C09108=1072.205,-104.494,443.420,172.641,21.693,153.924
C09109=1072.212,-104.245,443.411,172.643,21.694,153.924
C09110=1072.217,-103.995,443.400,172.644,21.695,153.924
C09111=1072.223,-103.745,443.390,172.646,21.696,153.924
C09112=1072.230,-103.495,443.381,172.648,21.697,153.924
C09113=1072.236,-103.246,443.370,172.649,21.699,153.924
C09114=1072.242,-102.996,443.360,172.651,21.700,153.924
C09115=1072.248,-102.746,443.351,172.652,21.701,153.924
C09116=1072.254,-102.497,443.340,172.654,21.702,153.924
C09117=1072.260,-102.247,443.330,172.656,21.704,153.924
C09118=1072.266,-101.997,443.321,172.657,21.705,153.924
C09119=1072.272,-101.748,443.310,172.659,21.706,153.924
C09120=1072.278,-101.498,443.301,172.660,21.708,153.924
C09121=1072.284,-101.249,443.290,172.662,21.709,153.924
C09122=1072.290,-100.999,443.280,172.663,21.710,153.924
C09123=1072.297,-100.748,443.270,172.664,21.711,153.924
C09124=1072.303,-100.499,443.259,172.666,21.712,153.924
C09125=1072.309,-100.249,443.250,172.668,21.714,153.924
C09126=1072.316,-100.000,443.240,172.669,21.715,153.924
C09127=1072.321,-99.750,443.229,172.671,21.716,153.924
C09128=1072.327,-99.500,443.220,172.672,21.717,153.924
C09129=1072.334,-99.251,443.210,172.674,21.719,153.924
C09130=1072.339,-99.001,443.199,172.676,21.720,153.924
C09131=1072.346,-98.752,443.189,172.677,21.721,153.924
C09132=1072.352,-98.501,443.179,172.679,21.722,153.924
C09133=1072.359,-98.220,443.167,172.681,21.724,153.924
C09134=1072.365,-97.938,443.156,172.683,21.726,153.924
C09135=1072.373,-97.657,443.145,172.685,21.727,153.924
C09136=1072.379,-97.374,443.133,172.686,21.728,153.924
C09137=1072.386,-97.125,443.123,172.688,21.730,153.924
C09138=1072.391,-96.875,443.113,172.689,21.731,153.924
C09139=1072.397,-96.626,443.102,172.691,21.733,153.924
C09140=1072.403,-96.376,443.093,172.692,21.734,153.924
C09141=1072.409,-96.126,443.082,172.694,21.735,153.924
C09142=1072.415,-95.877,443.071,172.696,21.737,153.924
C09143=1072.421,-95.626,443.061,172.697,21.738,153.924
C09144=1072.428,-95.377,443.051,172.699,21.739,153.924
C09145=1072.433,-95.127,443.040,172.700,21.741,153.924
C09146=1072.440,-94.878,443.030,172.702,21.742,153.924
C09147=1072.445,-94.628,443.020,172.703,21.744,153.924
C09148=1072.452,-94.379,443.010,172.705,21.745,153.924
C09149=1072.457,-94.128,443.000,172.707,21.746,153.924
C09150=1072.464,-93.879,442.989,172.708,21.748,153.924
C09151=1072.470,-93.629,442.978,172.710,21.749,153.924
C09152=1072.475,-93.379,442.968,172.711,21.751,153.924
C09153=1072.482,-93.130,442.958,172.713,21.753,153.924
C09154=1072.487,-92.880,442.947,172.714,21.754,153.924
C09155=1072.494,-92.630,442.937,172.716,21.755,153.924
C09156=1072.500,-92.381,442.926,172.717,21.757,153.924
C09157=1072.506,-92.131,442.917,172.719,21.758,153.924
C09158=1072.512,-91.881,442.905,172.721,21.759,153.924
C09159=1072.518,-91.631,442.895,172.722,21.761,153.924
C09160=1072.524,-91.382,442.885,172.724,21.762,153.924
C09161=1072.530,-91.132,442.874,172.725,21.764,153.924
C09162=1072.536,-90.882,442.865,172.727,21.765,153.924
C09163=1072.542,-90.632,442.853,172.728,21.766,153.924
C09164=1072.548,-90.383,442.842,172.730,21.768,153.924
C09165=1072.554,-90.133,442.833,172.731,21.770,153.924
C09166=1072.560,-89.883,442.822,172.733,21.771,153.924
C09167=1072.566,-89.634,442.812,172.735,21.773,153.924
C09168=1072.573,-89.384,442.800,172.736,21.774,153.924
C09169=1072.578,-89.134,442.790,172.738,21.775,153.924
C09170=1072.585,-88.885,442.780,172.739,21.777,153.924
C09171=1072.590,-88.635,442.769,172.741,21.778,153.924
C09172=1072.597,-88.386,442.760,172.742,21.780,153.925
C09173=1072.603,-88.135,442.748,172.744,21.781,153.925
C09174=1072.609,-87.886,442.737,172.745,21.783,153.925
C09175=1072.615,-87.637,442.727,172.747,21.784,153.925
C09176=1072.621,-87.387,442.717,172.748,21.786,153.925
C09177=1072.628,-87.137,442.706,172.750,21.787,153.925
C09178=1072.633,-86.887,442.695,172.751,21.789,153.925
C09179=1072.639,-86.638,442.685,172.753,21.790,153.925
C09180=1072.646,-86.389,442.674,172.755,21.792,153.925
C09181=1072.652,-86.138,442.664,172.756,21.793,153.925
C09182=1072.657,-85.888,442.653,172.758,21.794,153.925
C09183=1072.664,-85.639,442.643,172.759,21.796,153.925
C09184=1072.670,-85.389,442.631,172.761,21.798,153.925
C09185=1072.676,-85.139,442.620,172.762,21.799,153.925
C09186=1072.682,-84.890,442.611,172.764,21.801,153.925
C09187=1072.688,-84.640,442.600,172.765,21.802,153.925
C09188=1072.694,-84.390,442.589,172.767,21.804,153.925
C09189=1072.701,-84.141,442.579,172.768,21.805,153.925
C09190=1072.706,-83.891,442.568,172.770,21.807,153.925
C09191=1072.713,-83.641,442.556,172.772,21.808,153.925
C09192=1072.719,-83.392,442.546,172.773,21.809,153.925
C09193=1072.725,-83.142,442.536,172.774,21.811,153.926
C09194=1072.731,-82.892,442.525,172.776,21.813,153.926
C09195=1072.737,-82.642,442.514,172.778,21.814,153.926
C09196=1072.743,-82.393,442.504,172.779,21.816,153.926
C09197=1072.750,-82.113,442.492,172.781,21.817,153.926
C09198=1072.758,-81.834,442.480,172.783,21.819,153.926
C09199=1072.764,-81.554,442.467,172.784,21.821,153.926
C09200=1072.771,-81.275,442.455,172.786,21.823,153.926
C09201=1072.777,-81.026,442.444,172.788,21.824,153.926
C09202=1072.784,-80.776,442.434,172.789,21.826,153.926
C09203=1072.790,-80.526,442.423,172.791,21.827,153.926
C09204=1072.795,-80.277,442.412,172.792,21.829,153.926
C09205=1072.802,-80.027,442.401,172.793,21.831,153.926
C09206=1072.808,-79.778,442.390,172.795,21.832,153.926
C09207=1072.814,-79.527,442.380,172.797,21.833,153.926
C09208=1072.820,-79.277,442.369,172.798,21.835,153.926
C09209=1072.826,-79.028,442.358,172.800,21.837,153.926
C09210=1072.832,-78.778,442.347,172.801,21.839,153.927
C09211=1072.838,-78.528,442.336,172.803,21.840,153.927
C09212=1072.844,-78.279,442.325,172.804,21.842,153.927
C09213=1072.850,-78.030,442.313,172.805,21.843,153.927
C09214=1072.857,-77.780,442.303,172.807,21.845,153.927
C09215=1072.862,-77.530,442.292,172.809,21.847,153.927
C09216=1072.869,-77.280,442.281,172.811,21.848,153.927
C09217=1072.875,-77.031,442.270,172.812,21.850,153.927
C09218=1072.880,-76.781,442.259,172.814,21.852,153.927
C09219=1072.887,-76.531,442.248,172.815,21.854,153.927
C09220=1072.892,-76.281,442.237,172.817,21.855,153.927
C09221=1072.898,-76.032,442.226,172.818,21.857,153.927
C09222=1072.904,-75.782,442.215,172.820,21.858,153.927
C09223=1072.910,-75.532,442.204,172.821,21.860,153.928
C09224=1072.917,-75.282,442.193,172.823,21.862,153.928
C09225=1072.923,-75.033,442.182,172.824,21.864,153.928
C09226=1072.929,-74.783,442.171,172.826,21.865,153.928
C09227=1072.935,-74.534,442.159,172.827,21.867,153.928
C09228=1072.941,-74.284,442.149,172.829,21.868,153.928
C09229=1072.947,-74.034,442.137,172.830,21.870,153.928
C09230=1072.953,-73.785,442.126,172.832,21.872,153.928
C09231=1072.959,-73.535,442.116,172.833,21.874,153.928
C09232=1072.965,-73.285,442.104,172.835,21.875,153.928
C09233=1072.970,-73.035,442.093,172.836,21.877,153.928
C09234=1072.976,-72.786,442.081,172.837,21.879,153.929
C09235=1072.983,-72.536,442.070,172.839,21.880,153.929
C09236=1072.988,-72.287,442.059,172.840,21.882,153.929
C09237=1072.994,-72.037,442.048,172.842,21.884,153.929
C09238=1073.000,-71.787,442.037,172.843,21.886,153.929
C09239=1073.007,-71.538,442.025,172.845,21.888,153.929
C09240=1073.012,-71.288,442.014,172.847,21.890,153.929
C09241=1073.018,-71.038,442.003,172.848,21.891,153.929
C09242=1073.024,-70.789,441.992,172.850,21.893,153.929
C09243=1073.030,-70.538,441.981,172.851,21.895,153.930
C09244=1073.036,-70.290,441.969,172.853,21.897,153.930
C09245=1073.042,-70.039,441.958,172.854,21.898,153.930
C09246=1073.048,-69.790,441.947,172.856,21.900,153.930
C09247=1073.053,-69.540,441.935,172.857,21.902,153.930
C09248=1073.060,-69.291,441.923,172.859,21.904,153.930
C09249=1073.065,-69.041,441.913,172.860,21.906,153.930
C09250=1073.072,-68.791,441.901,172.861,21.908,153.930
C09251=1073.078,-68.542,441.890,172.863,21.909,153.930
C09252=1073.084,-68.292,441.878,172.864,21.911,153.930
C09253=1073.089,-68.042,441.867,172.866,21.913,153.931
C09254=1073.095,-67.792,441.856,172.867,21.914,153.931
C09255=1073.102,-67.543,441.844,172.869,21.916,153.931
C09256=1073.107,-67.293,441.833,172.870,21.918,153.931
C09257=1073.114,-67.043,441.822,172.871,21.920,153.931
C09258=1073.119,-66.794,441.810,172.873,21.921,153.931
C09259=1073.125,-66.544,441.799,172.875,21.924,153.931
C09260=1073.131,-66.295,441.787,172.877,21.926,153.931
C09261=1073.138,-66.018,441.774,172.878,21.928,153.932
C09262=1073.145,-65.740,441.762,172.879,21.930,153.932
C09263=1073.152,-65.463,441.750,172.881,21.931,153.932
C09264=1073.158,-65.185,441.736,172.883,21.934,153.932
C09265=1073.164,-64.937,441.725,172.885,21.935,153.932
C09266=1073.170,-64.686,441.714,172.886,21.937,153.932
C09267=1073.176,-64.438,441.702,172.887,21.939,153.932
C09268=1073.182,-64.187,441.690,172.889,21.941,153.932
C09269=1073.188,-63.937,441.679,172.890,21.943,153.933
C09270=1073.194,-63.688,441.667,172.892,21.944,153.933
C09271=1073.200,-63.438,441.656,172.893,21.946,153.933
C09272=1073.206,-63.189,441.644,172.895,21.948,153.933
C09273=1073.212,-62.938,441.633,172.896,21.950,153.933
C09274=1073.218,-62.689,441.621,172.897,21.952,153.933
C09275=1073.224,-62.439,441.610,172.899,21.953,153.933
C09276=1073.230,-62.190,441.598,172.900,21.955,153.933
C09277=1073.236,-61.940,441.586,172.903,21.958,153.933
C09278=1073.242,-61.691,441.575,172.904,21.960,153.934
C09279=1073.248,-61.441,441.564,172.905,21.962,153.934
C09280=1073.254,-61.192,441.552,172.907,21.963,153.934
C09281=1073.260,-60.941,441.540,172.908,21.965,153.934
C09282=1073.267,-60.692,441.528,172.910,21.967,153.934
C09283=1073.272,-60.442,441.517,172.911,21.969,153.934
C09284=1073.279,-60.193,441.505,172.912,21.971,153.934
C09285=1073.284,-59.943,441.494,172.914,21.973,153.935
C09286=1073.291,-59.693,441.482,172.915,21.974,153.935
C09287=1073.297,-59.443,441.471,172.917,21.976,153.935
C09288=1073.302,-59.194,441.458,172.918,21.978,153.935
C09289=1073.309,-58.944,441.447,172.920,21.980,153.935
C09290=1073.315,-58.695,441.436,172.921,21.982,153.935
C09291=1073.321,-58.445,441.424,172.923,21.984,153.935
C09292=1073.327,-58.195,441.412,172.925,21.986,153.935
C09293=1073.333,-57.946,441.400,172.926,21.987,153.935
C09294=1073.339,-57.696,441.389,172.928,21.989,153.936
C09295=1073.345,-57.446,441.376,172.929,21.991,153.936
C09296=1073.351,-57.197,441.365,172.930,21.993,153.936
C09297=1073.358,-56.947,441.354,172.932,21.995,153.936
C09298=1073.363,-56.698,441.341,172.933,21.997,153.936
C09299=1073.369,-56.448,441.330,172.935,21.999,153.936
C09300=1073.376,-56.198,441.318,172.936,22.001,153.937
C09301=1073.382,-55.949,441.307,172.937,22.002,153.937
C09302=1073.388,-55.699,441.295,172.939,22.004,153.937
C09303=1073.394,-55.449,441.283,172.940,22.006,153.937
C09304=1073.400,-55.200,441.271,172.942,22.008,153.937
C09305=1073.406,-54.950,441.259,172.944,22.010,153.937
C09306=1073.413,-54.700,441.247,172.945,22.012,153.937
C09307=1073.419,-54.451,441.236,172.947,22.014,153.937
C09308=1073.425,-54.201,441.223,172.948,22.016,153.938
C09309=1073.431,-53.951,441.212,172.949,22.018,153.938
C09310=1073.438,-53.702,441.200,172.951,22.020,153.938
C09311=1073.443,-53.452,441.188,172.952,22.022,153.938
C09312=1073.449,-53.202,441.177,172.954,22.024,153.938
C09313=1073.456,-52.953,441.165,172.955,22.025,153.938
C09314=1073.461,-52.703,441.153,172.957,22.027,153.938
C09315=1073.468,-52.454,441.141,172.958,22.029,153.939
C09316=1073.473,-52.203,441.129,172.959,22.031,153.939
C09317=1073.480,-51.954,441.117,172.962,22.033,153.939
C09318=1073.486,-51.705,441.105,172.963,22.035,153.939
C09319=1073.492,-51.455,441.093,172.964,22.037,153.939
C09320=1073.499,-51.206,441.081,172.966,22.039,153.939
C09321=1073.505,-50.955,441.069,172.967,22.041,153.939
C09322=1073.510,-50.706,441.057,172.969,22.043,153.940
C09323=1073.517,-50.457,441.045,172.970,22.045,153.940
C09324=1073.523,-50.207,441.033,172.971,22.047,153.940
C09325=1073.529,-49.931,441.020,172.973,22.049,153.940
C09326=1073.536,-49.655,441.006,172.975,22.052,153.940
C09327=1073.543,-49.379,440.993,172.976,22.054,153.940
C09328=1073.549,-49.103,440.979,172.978,22.056,153.941
C09329=1073.555,-48.854,440.967,172.979,22.058,153.941
C09330=1073.561,-48.604,440.956,172.981,22.060,153.941
C09331=1073.567,-48.354,440.944,172.983,22.062,153.941
C09332=1073.573,-48.105,440.931,172.984,22.064,153.941
C09333=1073.579,-47.855,440.919,172.985,22.066,153.941
C09334=1073.585,-47.605,440.907,172.987,22.068,153.942
C09335=1073.591,-47.356,440.894,172.988,22.070,153.942
C09336=1073.597,-47.106,440.882,172.989,22.072,153.942
C09337=1073.603,-46.857,440.870,172.991,22.074,153.942
C09338=1073.609,-46.607,440.858,172.992,22.076,153.942
C09339=1073.614,-46.358,440.845,172.993,22.078,153.942
C09340=1073.621,-46.108,440.833,172.995,22.080,153.943
C09341=1073.627,-45.858,440.821,172.997,22.083,153.943
C09342=1073.633,-45.608,440.809,172.998,22.085,153.943
C09343=1073.639,-45.359,440.797,173.000,22.087,153.943
C09344=1073.644,-45.109,440.785,173.001,22.089,153.943
C09345=1073.650,-44.859,440.772,173.003,22.091,153.943
C09346=1073.657,-44.610,440.760,173.004,22.093,153.944
C09347=1073.662,-44.360,440.748,173.005,22.095,153.944
C09348=1073.668,-44.111,440.736,173.007,22.097,153.944
C09349=1073.675,-43.861,440.724,173.008,22.099,153.944
C09350=1073.681,-43.611,440.711,173.009,22.101,153.944
C09351=1073.687,-43.361,440.699,173.012,22.103,153.944
C09352=1073.692,-43.112,440.686,173.013,22.106,153.945
C09353=1073.699,-42.862,440.674,173.014,22.108,153.945
C09354=1073.705,-42.613,440.661,173.016,22.110,153.945
C09355=1073.711,-42.363,440.649,173.017,22.112,153.945
C09356=1073.717,-42.114,440.637,173.018,22.113,153.945
C09357=1073.723,-41.865,440.624,173.020,22.116,153.946
C09358=1073.729,-41.615,440.612,173.021,22.118,153.946
C09359=1073.735,-41.365,440.599,173.022,22.120,153.946
C09360=1073.741,-41.115,440.587,173.024,22.122,153.946
C09361=1073.747,-40.865,440.575,173.026,22.124,153.946
C09362=1073.752,-40.616,440.563,173.027,22.126,153.947
C09363=1073.759,-40.367,440.551,173.029,22.128,153.947
C09364=1073.765,-40.117,440.538,173.030,22.130,153.947
C09365=1073.771,-39.867,440.525,173.031,22.132,153.947
C09366=1073.777,-39.618,440.512,173.033,22.135,153.947
C09367=1073.784,-39.368,440.500,173.034,22.137,153.947
C09368=1073.790,-39.118,440.488,173.035,22.139,153.948
C09369=1073.795,-38.869,440.476,173.037,22.140,153.948
C09370=1073.801,-38.619,440.463,173.038,22.143,153.948
C09371=1073.807,-38.369,440.451,173.040,22.145,153.948
C09372=1073.814,-38.120,440.438,173.042,22.147,153.948
C09373=1073.820,-37.870,440.425,173.043,22.150,153.949
C09374=1073.826,-37.620,440.413,173.044,22.152,153.949
C09375=1073.831,-37.371,440.401,173.046,22.154,153.949
C09376=1073.837,-37.121,440.388,173.047,22.156,153.949
C09377=1073.843,-36.872,440.375,173.048,22.158,153.949
C09378=1073.849,-36.622,440.362,173.050,22.160,153.949
C09379=1073.855,-36.372,440.350,173.051,22.162,153.950
C09380=1073.861,-36.122,440.337,173.053,22.165,153.950
C09381=1073.866,-35.873,440.325,173.054,22.167,153.950
C09382=1073.872,-35.624,440.312,173.056,22.169,153.950
C09383=1073.878,-35.374,440.299,173.057,22.171,153.950
C09384=1073.884,-35.124,440.287,173.058,22.173,153.951
C09385=1073.890,-34.875,440.273,173.060,22.175,153.951
C09386=1073.896,-34.625,440.261,173.061,22.177,153.951
C09387=1073.903,-34.375,440.249,173.062,22.180,153.951
C09388=1073.909,-34.126,440.236,173.064,22.182,153.951
C09389=1073.915,-33.851,440.221,173.066,22.185,153.952
C09390=1073.922,-33.575,440.208,173.067,22.186,153.952
C09391=1073.928,-33.300,440.194,173.068,22.189,153.952
C09392=1073.935,-33.024,440.180,173.071,22.192,153.952
C09393=1073.941,-32.775,440.167,173.072,22.194,153.953
C09394=1073.947,-32.525,440.154,173.073,22.196,153.953
C09395=1073.953,-32.275,440.142,173.075,22.198,153.953
C09396=1073.959,-32.026,440.128,173.076,22.200,153.953
C09397=1073.965,-31.776,440.116,173.077,22.203,153.953
C09398=1073.971,-31.526,440.103,173.079,22.204,153.954
C09399=1073.977,-31.277,440.090,173.081,22.207,153.954
C09400=1073.983,-31.027,440.077,173.082,22.209,153.954
C09401=1073.989,-30.777,440.065,173.083,22.211,153.954
C09402=1073.995,-30.528,440.052,173.085,22.214,153.954
C09403=1074.001,-30.278,440.039,173.086,22.216,153.955
C09404=1074.007,-30.029,440.026,173.087,22.218,153.955
C09405=1074.013,-29.779,440.013,173.089,22.220,153.955
C09406=1074.019,-29.530,440.000,173.090,22.222,153.955
C09407=1074.024,-29.280,439.988,173.091,22.224,153.955
C09408=1074.030,-29.030,439.975,173.094,22.227,153.956
C09409=1074.037,-28.781,439.962,173.095,22.229,153.956
C09410=1074.042,-28.531,439.949,173.096,22.231,153.956
C09411=1074.049,-28.282,439.936,173.097,22.233,153.956
C09412=1074.055,-28.032,439.924,173.099,22.235,153.956
C09413=1074.061,-27.783,439.910,173.100,22.238,153.957
C09414=1074.067,-27.533,439.898,173.101,22.240,153.957
C09415=1074.073,-27.284,439.885,173.103,22.242,153.957
C09416=1074.079,-27.034,439.872,173.104,22.244,153.957
C09417=1074.084,-26.784,439.858,173.106,22.246,153.957
C09418=1074.090,-26.534,439.846,173.108,22.249,153.958
C09419=1074.096,-26.285,439.832,173.109,22.251,153.958
C09420=1074.102,-26.035,439.820,173.110,22.253,153.958
C09421=1074.109,-25.786,439.806,173.111,22.256,153.958
C09422=1074.114,-25.536,439.793,173.113,22.258,153.959
C09423=1074.120,-25.287,439.780,173.114,22.260,153.959
C09424=1074.126,-25.037,439.767,173.115,22.262,153.959
C09425=1074.132,-24.787,439.754,173.117,22.265,153.959
C09426=1074.138,-24.538,439.740,173.119,22.267,153.959
C09427=1074.143,-24.288,439.728,173.120,22.269,153.960
C09428=1074.150,-24.039,439.715,173.121,22.272,153.960
C09429=1074.156,-23.789,439.701,173.123,22.274,153.960
C09430=1074.162,-23.540,439.689,173.124,22.276,153.960
C09431=1074.167,-23.290,439.675,173.125,22.278,153.961
C09432=1074.173,-23.040,439.662,173.127,22.281,153.961
C09433=1074.179,-22.791,439.649,173.129,22.283,153.961
C09434=1074.186,-22.542,439.636,173.130,22.285,153.961
C09435=1074.191,-22.291,439.623,173.131,22.288,153.962
C09436=1074.197,-22.042,439.609,173.133,22.290,153.962
C09437=1074.203,-21.793,439.596,173.134,22.292,153.962
C09438=1074.208,-21.543,439.583,173.135,22.294,153.962
C09439=1074.215,-21.293,439.569,173.137,22.297,153.963
C09440=1074.221,-21.043,439.556,173.138,22.298,153.963
C09441=1074.227,-20.794,439.543,173.140,22.301,153.963
C09442=1074.233,-20.544,439.530,173.141,22.304,153.963
C09443=1074.239,-20.295,439.516,173.143,22.306,153.963
C09444=1074.245,-20.045,439.504,173.144,22.308,153.964
C09445=1074.251,-19.796,439.491,173.145,22.310,153.964
C09446=1074.257,-19.546,439.477,173.146,22.313,153.964
C09447=1074.263,-19.297,439.463,173.148,22.315,153.964
C09448=1074.269,-19.047,439.451,173.149,22.317,153.965
C09449=1074.274,-18.797,439.437,173.151,22.320,153.965
C09450=1074.280,-18.548,439.424,173.153,22.322,153.965
C09451=1074.287,-18.299,439.410,173.154,22.324,153.965
C09452=1074.292,-18.048,439.397,173.155,22.327,153.965
C09453=1074.299,-17.772,439.382,173.156,22.329,153.966
C09454=1074.306,-17.496,439.367,173.159,22.331,153.966
C09455=1074.313,-17.219,439.353,173.160,22.334,153.966
C09456=1074.319,-16.943,439.338,173.161,22.336,153.966
C09457=1074.325,-16.694,439.325,173.162,22.339,153.967
C09458=1074.331,-16.444,439.311,173.165,22.341,153.967
C09459=1074.337,-16.195,439.298,173.166,22.344,153.967
C09460=1074.343,-15.946,439.284,173.167,22.346,153.967
C09461=1074.349,-15.695,439.270,173.168,22.348,153.968
C09462=1074.355,-15.445,439.258,173.170,22.350,153.968
C09463=1074.362,-15.196,439.244,173.171,22.352,153.968
C09464=1074.367,-14.947,439.231,173.172,22.355,153.968
C09465=1074.373,-14.697,439.217,173.174,22.358,153.969
C09466=1074.379,-14.448,439.203,173.176,22.360,153.969
C09467=1074.385,-14.198,439.190,173.177,22.362,153.969
C09468=1074.390,-13.949,439.176,173.178,22.364,153.969
C09469=1074.397,-13.699,439.163,173.179,22.367,153.970
C09470=1074.403,-13.449,439.149,173.181,22.369,153.970
C09471=1074.409,-13.199,439.136,173.182,22.371,153.970
C09472=1074.414,-12.950,439.122,173.183,22.374,153.970
C09473=1074.420,-12.701,439.109,173.185,22.377,153.971
C09474=1074.426,-12.451,439.095,173.187,22.379,153.971
C09475=1074.432,-12.202,439.082,173.188,22.381,153.971
C09476=1074.438,-11.952,439.068,173.189,22.383,153.971
C09477=1074.444,-11.702,439.054,173.191,22.385,153.971
C09478=1074.450,-11.453,439.041,173.192,22.388,153.972
C09479=1074.455,-11.203,439.027,173.193,22.390,153.972
C09480=1074.461,-10.954,439.013,173.195,22.393,153.972
C09481=1074.467,-10.704,439.000,173.197,22.395,153.972
C09482=1074.474,-10.454,438.986,173.198,22.397,153.973
C09483=1074.479,-10.205,438.972,173.199,22.400,153.973
C09484=1074.485,-9.955,438.959,173.200,22.402,153.973
C09485=1074.491,-9.706,438.945,173.202,22.404,153.973
C09486=1074.497,-9.457,438.932,173.203,22.407,153.974
C09487=1074.503,-9.206,438.917,173.204,22.409,153.974
C09488=1074.509,-8.957,438.904,173.206,22.412,153.974
C09489=1074.515,-8.708,438.890,173.208,22.414,153.974
C09490=1074.520,-8.458,438.876,173.209,22.416,153.975
C09491=1074.527,-8.209,438.863,173.210,22.419,153.975
C09492=1074.533,-7.959,438.848,173.211,22.421,153.975
C09493=1074.539,-7.710,438.835,173.213,22.423,153.975
C09494=1074.545,-7.460,438.821,173.214,22.426,153.976
C09495=1074.550,-7.211,438.807,173.216,22.429,153.976
C09496=1074.557,-6.961,438.794,173.217,22.431,153.976
C09497=1074.562,-6.711,438.780,173.219,22.433,153.976
C09498=1074.569,-6.462,438.766,173.220,22.435,153.977
C09499=1074.574,-6.212,438.753,173.221,22.438,153.977
C09500=1074.580,-5.962,438.738,173.223,22.440,153.977
C09501=1074.587,-5.713,438.724,173.224,22.442,153.977
C09502=1074.592,-5.464,438.711,173.226,22.445,153.978
C09503=1074.598,-5.214,438.697,173.227,22.447,153.978
C09504=1074.604,-4.964,438.683,173.228,22.449,153.978
C09505=1074.610,-4.715,438.669,173.230,22.452,153.978
C09506=1074.616,-4.465,438.656,173.231,22.454,153.979
C09507=1074.623,-4.216,438.641,173.232,22.457,153.979
C09508=1074.629,-3.966,438.628,173.234,22.459,153.979
C09509=1074.634,-3.717,438.614,173.236,22.461,153.979
C09510=1074.640,-3.467,438.600,173.237,22.464,153.980
C09511=1074.647,-3.217,438.586,173.238,22.466,153.980
C09512=1074.652,-2.968,438.572,173.239,22.469,153.980
C09513=1074.658,-2.719,438.558,173.241,22.471,153.981
C09514=1074.664,-2.468,438.544,173.242,22.473,153.981
C09515=1074.669,-2.219,438.530,173.243,22.476,153.981
C09516=1074.675,-1.970,438.515,173.245,22.479,153.981
C09517=1074.681,-1.692,438.500,173.247,22.481,153.982
C09518=1074.688,-1.414,438.485,173.248,22.484,153.982
C09519=1074.694,-1.136,438.469,173.250,22.487,153.982
C09520=1074.701,-0.858,438.453,173.251,22.489,153.982
C09521=1074.707,-0.608,438.439,173.252,22.492,153.983
C09522=1074.712,-0.359,438.424,173.253,22.494,153.983
C09523=1074.719,-0.109,438.411,173.256,22.497,153.983
C09524=1074.725,0.140,438.397,173.257,22.499,153.984
C09525=1074.730,0.390,438.383,173.258,22.502,153.984
C09526=1074.737,0.639,438.368,173.259,22.504,153.984
C09527=1074.742,0.889,438.354,173.261,22.506,153.984
C09528=1074.748,1.138,438.339,173.262,22.509,153.985
C09529=1074.753,1.387,438.326,173.263,22.511,153.985
C09530=1074.759,1.638,438.311,173.265,22.514,153.985
C09531=1074.765,1.887,438.297,173.266,22.516,153.985
C09532=1074.771,2.136,438.283,173.268,22.519,153.986
C09533=1074.777,2.386,438.269,173.269,22.521,153.986
C09534=1074.783,2.635,438.255,173.270,22.524,153.986
C09535=1074.789,2.885,438.241,173.272,22.526,153.986
C09536=1074.795,3.134,438.226,173.273,22.528,153.987
C09537=1074.801,3.384,438.212,173.275,22.531,153.987
C09538=1074.806,3.633,438.197,173.276,22.533,153.987
C09539=1074.812,3.883,438.183,173.277,22.536,153.988
C09540=1074.818,4.133,438.169,173.279,22.538,153.988
C09541=1074.824,4.382,438.155,173.280,22.541,153.988
C09542=1074.830,4.632,438.141,173.281,22.543,153.988
C09543=1074.836,4.881,438.126,173.282,22.546,153.989
C09544=1074.842,5.131,438.112,173.284,22.549,153.989
C09545=1074.847,5.380,438.097,173.286,22.550,153.989
C09546=1074.854,5.629,438.084,173.287,22.553,153.989
C09547=1074.860,5.879,438.069,173.288,22.555,153.990
C09548=1074.866,6.129,438.055,173.290,22.558,153.990
C09549=1074.872,6.378,438.040,173.291,22.560,153.990
C09550=1074.877,6.628,438.026,173.293,22.563,153.991
C09551=1074.883,6.877,438.012,173.294,22.566,153.991
C09552=1074.889,7.127,437.997,173.295,22.568,153.991
C09553=1074.895,7.376,437.983,173.297,22.570,153.991
C09554=1074.901,7.626,437.969,173.298,22.572,153.992
C09555=1074.907,7.875,437.954,173.299,22.575,153.992
C09556=1074.913,8.124,437.940,173.301,22.577,153.992
C09557=1074.919,8.375,437.925,173.303,22.580,153.992
C09558=1074.925,8.624,437.911,173.304,22.582,153.993
C09559=1074.931,8.874,437.896,173.305,22.585,153.993
C09560=1074.936,9.123,437.882,173.306,22.587,153.993
C09561=1074.943,9.372,437.867,173.308,22.590,153.994
C09562=1074.948,9.622,437.853,173.309,22.592,153.994
C09563=1074.955,9.872,437.838,173.310,22.594,153.994
C09564=1074.960,10.121,437.824,173.312,22.597,153.994
C09565=1074.966,10.371,437.809,173.314,22.599,153.994
C09566=1074.972,10.620,437.795,173.315,22.602,153.995
C09567=1074.978,10.870,437.781,173.316,22.604,153.995
C09568=1074.984,11.119,437.766,173.317,22.607,153.995
C09569=1074.990,11.369,437.751,173.319,22.609,153.996
C09570=1074.996,11.618,437.737,173.321,22.612,153.996
C09571=1075.002,11.868,437.722,173.322,22.615,153.996
C09572=1075.008,12.117,437.708,173.323,22.616,153.996
C09573=1075.014,12.367,437.693,173.325,22.619,153.997
C09574=1075.020,12.616,437.679,173.326,22.621,153.997
C09575=1075.026,12.866,437.664,173.327,22.624,153.997
C09576=1075.032,13.115,437.649,173.329,22.627,153.997
C09577=1075.038,13.365,437.635,173.330,22.629,153.998
C09578=1075.044,13.614,437.620,173.332,22.631,153.998
C09579=1075.050,13.864,437.606,173.333,22.634,153.998
C09580=1075.056,14.113,437.591,173.334,22.636,153.998
C09581=1075.063,14.393,437.574,173.336,22.639,153.999
C09582=1075.069,14.673,437.558,173.338,22.642,153.999
C09583=1075.076,14.953,437.542,173.339,22.644,153.999
C09584=1075.082,15.233,437.525,173.341,22.647,154.000
C09585=1075.088,15.483,437.510,173.342,22.650,154.000
C09586=1075.094,15.732,437.496,173.343,22.652,154.000
C09587=1075.100,15.981,437.481,173.344,22.655,154.001
C09588=1075.106,16.230,437.466,173.346,22.657,154.001
C09589=1075.112,16.481,437.451,173.348,22.660,154.001
C09590=1075.117,16.730,437.437,173.349,22.662,154.002
C09591=1075.124,16.979,437.422,173.350,22.665,154.002
C09592=1075.129,17.228,437.407,173.352,22.667,154.002
C09593=1075.135,17.478,437.392,173.353,22.670,154.002
C09594=1075.141,17.727,437.377,173.354,22.672,154.003
C09595=1075.147,17.977,437.362,173.356,22.675,154.003
C09596=1075.153,18.227,437.348,173.358,22.677,154.003
C09597=1075.158,18.477,437.333,173.359,22.679,154.003
C09598=1075.165,18.726,437.318,173.360,22.682,154.004
C09599=1075.171,18.975,437.303,173.361,22.684,154.004
C09600=1075.177,19.225,437.288,173.363,22.687,154.004
C09601=1075.182,19.474,437.273,173.365,22.690,154.004
C09602=1075.188,19.724,437.258,173.366,22.692,154.005
C09603=1075.194,19.973,437.243,173.367,22.694,154.005
C09604=1075.200,20.223,437.228,173.368,22.697,154.005
C09605=1075.206,20.472,437.213,173.370,22.699,154.006
C09606=1075.212,20.721,437.198,173.371,22.702,154.006
C09607=1075.218,20.971,437.183,173.373,22.705,154.006
C09608=1075.223,21.220,437.168,173.374,22.707,154.006
C09609=1075.230,21.470,437.153,173.376,22.709,154.007
C09610=1075.235,21.719,437.138,173.377,22.712,154.007
C09611=1075.241,21.969,437.123,173.378,22.714,154.007
C09612=1075.247,22.219,437.108,173.379,22.717,154.008
C09613=1075.253,22.468,437.093,173.381,22.720,154.008
C09614=1075.259,22.717,437.078,173.383,22.722,154.008
C09615=1075.264,22.967,437.063,173.384,22.724,154.008
C09616=1075.270,23.216,437.048,173.385,22.727,154.009
C09617=1075.277,23.466,437.033,173.386,22.729,154.009
C09618=1075.282,23.715,437.018,173.388,22.732,154.009
C09619=1075.288,23.965,437.003,173.390,22.735,154.010
C09620=1075.293,24.214,436.988,173.391,22.737,154.010
C09621=1075.300,24.464,436.973,173.392,22.739,154.010
C09622=1075.305,24.714,436.957,173.394,22.742,154.010
C09623=1075.311,24.963,436.943,173.395,22.744,154.011
C09624=1075.317,25.212,436.928,173.397,22.747,154.011
C09625=1075.323,25.462,436.912,173.398,22.750,154.011
C09626=1075.329,25.711,436.897,173.399,22.752,154.012
C09627=1075.335,25.961,436.881,173.401,22.754,154.012
C09628=1075.341,26.210,436.866,173.402,22.757,154.012
C09629=1075.347,26.459,436.852,173.403,22.759,154.012
C09630=1075.353,26.709,436.836,173.405,22.762,154.013
C09631=1075.359,26.959,436.821,173.407,22.765,154.013
C09632=1075.364,27.208,436.806,173.408,22.767,154.013
C09633=1075.371,27.457,436.790,173.409,22.769,154.014
C09634=1075.376,27.707,436.775,173.410,22.772,154.014
C09635=1075.382,27.956,436.760,173.412,22.774,154.014
C09636=1075.388,28.206,436.745,173.414,22.777,154.014
C09637=1075.394,28.456,436.730,173.415,22.780,154.015
C09638=1075.400,28.704,436.714,173.416,22.782,154.015
C09639=1075.406,28.954,436.699,173.417,22.784,154.015
C09640=1075.412,29.204,436.683,173.418,22.787,154.016
C09641=1075.417,29.453,436.668,173.421,22.790,154.016
C09642=1075.423,29.702,436.653,173.422,22.793,154.016
C09643=1075.429,29.952,436.637,173.423,22.795,154.016
C09644=1075.435,30.201,436.623,173.424,22.798,154.017
C09645=1075.441,30.483,436.605,173.427,22.800,154.017
C09646=1075.448,30.764,436.587,173.428,22.803,154.017
C09647=1075.455,31.045,436.570,173.429,22.806,154.018
C09648=1075.460,31.326,436.552,173.431,22.809,154.018
C09649=1075.467,31.576,436.537,173.432,22.812,154.018
C09650=1075.473,31.826,436.522,173.433,22.814,154.019
C09651=1075.479,32.075,436.506,173.435,22.816,154.019
C09652=1075.484,32.324,436.491,173.437,22.819,154.019
C09653=1075.490,32.574,436.476,173.438,22.822,154.020
C09654=1075.497,32.823,436.460,173.439,22.824,154.020
C09655=1075.502,33.073,436.445,173.440,22.827,154.020
C09656=1075.507,33.323,436.429,173.442,22.829,154.020
C09657=1075.514,33.572,436.414,173.444,22.832,154.021
C09658=1075.520,33.822,436.398,173.445,22.834,154.021
C09659=1075.525,34.070,436.382,173.446,22.837,154.021
C09660=1075.531,34.320,436.367,173.448,22.839,154.022
C09661=1075.537,34.570,436.352,173.449,22.842,154.022
C09662=1075.543,34.819,436.335,173.451,22.844,154.022
C09663=1075.549,35.068,436.321,173.452,22.847,154.022
C09664=1075.555,35.318,436.305,173.454,22.849,154.023
C09665=1075.560,35.568,436.289,173.455,22.852,154.023
C09666=1075.567,35.817,436.274,173.456,22.854,154.023
C09667=1075.572,36.066,436.258,173.458,22.857,154.023
C09668=1075.578,36.316,436.243,173.459,22.859,154.024
C09669=1075.584,36.565,436.227,173.461,22.862,154.024
C09670=1075.590,36.815,436.211,173.462,22.864,154.024
C09671=1075.596,37.064,436.195,173.463,22.867,154.025
C09672=1075.601,37.313,436.180,173.464,22.869,154.025
C09673=1075.608,37.562,436.164,173.467,22.872,154.025
C09674=1075.613,37.812,436.149,173.468,22.874,154.025
C09675=1075.619,38.062,436.132,173.469,22.877,154.026
C09676=1075.625,38.312,436.117,173.470,22.880,154.026
C09677=1075.631,38.560,436.102,173.471,22.882,154.026
C09678=1075.637,38.810,436.086,173.474,22.885,154.027
C09679=1075.643,39.059,436.070,173.475,22.887,154.027
C09680=1075.648,39.309,436.054,173.476,22.890,154.027
C09681=1075.654,39.559,436.038,173.477,22.892,154.028
C09682=1075.659,39.808,436.023,173.479,22.895,154.028
C09683=1075.665,40.057,436.007,173.481,22.897,154.028
C09684=1075.672,40.306,435.991,173.482,22.900,154.028
C09685=1075.678,40.556,435.975,173.483,22.902,154.029
C09686=1075.683,40.806,435.959,173.485,22.905,154.029
C09687=1075.689,41.055,435.944,173.486,22.908,154.029
C09688=1075.694,41.304,435.928,173.488,22.910,154.030
C09689=1075.700,41.554,435.911,173.489,22.913,154.030
C09690=1075.706,41.804,435.896,173.490,22.915,154.030
C09691=1075.712,42.053,435.880,173.492,22.918,154.031
C09692=1075.718,42.302,435.863,173.493,22.920,154.031
C09693=1075.724,42.551,435.849,173.495,22.923,154.031
C09694=1075.730,42.801,435.833,173.496,22.925,154.031
C09695=1075.735,43.051,435.817,173.498,22.928,154.032
C09696=1075.741,43.300,435.801,173.499,22.930,154.032
C09697=1075.747,43.549,435.785,173.500,22.933,154.032
C09698=1075.753,43.799,435.768,173.502,22.936,154.032
C09699=1075.759,44.049,435.753,173.503,22.938,154.033
C09700=1075.764,44.297,435.737,173.505,22.941,154.033
C09701=1075.770,44.547,435.721,173.506,22.943,154.033
C09702=1075.776,44.797,435.705,173.508,22.946,154.034
C09703=1075.782,45.046,435.689,173.509,22.949,154.034
C09704=1075.788,45.295,435.673,173.511,22.951,154.034
C09705=1075.792,45.544,435.656,173.512,22.953,154.035
C09706=1075.798,45.794,435.641,173.513,22.956,154.035
C09707=1075.804,46.044,435.624,173.515,22.959,154.035
C09708=1075.810,46.293,435.608,173.516,22.962,154.036
C09709=1075.816,46.575,435.590,173.518,22.964,154.036
C09710=1075.822,46.855,435.572,173.520,22.967,154.036
C09711=1075.829,47.137,435.554,173.521,22.970,154.037
C09712=1075.836,47.418,435.535,173.523,22.973,154.037
C09713=1075.841,47.668,435.519,173.524,22.976,154.037
C09714=1075.847,47.918,435.503,173.525,22.978,154.037
C09715=1075.853,48.167,435.487,173.527,22.980,154.038
C09716=1075.858,48.415,435.471,173.529,22.983,154.038
C09717=1075.864,48.665,435.455,173.530,22.986,154.038
C09718=1075.870,48.914,435.438,173.531,22.989,154.039
C09719=1075.876,49.164,435.422,173.532,22.991,154.039
C09720=1075.882,49.413,435.406,173.534,22.993,154.039
C09721=1075.887,49.663,435.390,173.536,22.996,154.040
C09722=1075.893,49.913,435.374,173.537,22.999,154.040
C09723=1075.899,50.162,435.357,173.538,23.001,154.040
C09724=1075.905,50.411,435.341,173.540,23.003,154.040
C09725=1075.911,50.661,435.325,173.542,23.006,154.041
C09726=1075.917,50.910,435.309,173.543,23.009,154.041
C09727=1075.922,51.160,435.292,173.544,23.011,154.041
C09728=1075.927,51.408,435.276,173.545,23.014,154.042
C09729=1075.933,51.658,435.260,173.547,23.017,154.042
C09730=1075.939,51.907,435.243,173.549,23.019,154.042
C09731=1075.945,52.156,435.227,173.550,23.022,154.043
C09732=1075.951,52.406,435.211,173.551,23.024,154.043
C09733=1075.956,52.655,435.194,173.553,23.027,154.043
C09734=1075.962,52.905,435.178,173.555,23.029,154.043
C09735=1075.968,53.154,435.161,173.556,23.032,154.044
C09736=1075.974,53.403,435.145,173.557,23.034,154.044
C09737=1075.980,53.653,435.129,173.559,23.037,154.044
C09738=1075.985,53.902,435.112,173.560,23.039,154.045
C09739=1075.991,54.152,435.096,173.562,23.042,154.045
C09740=1075.997,54.401,435.080,173.563,23.044,154.045
C09741=1076.003,54.650,435.063,173.565,23.047,154.045
C09742=1076.009,54.900,435.047,173.566,23.049,154.046
C09743=1076.014,55.149,435.030,173.568,23.052,154.046
C09744=1076.020,55.399,435.014,173.569,23.055,154.046
C09745=1076.026,55.648,434.998,173.570,23.057,154.047
C09746=1076.032,55.897,434.981,173.572,23.060,154.047
C09747=1076.038,56.147,434.965,173.574,23.063,154.047
C09748=1076.043,56.396,434.948,173.575,23.065,154.047
C09749=1076.049,56.646,434.932,173.576,23.067,154.048
C09750=1076.055,56.895,434.916,173.578,23.070,154.048
C09751=1076.062,57.145,434.899,173.579,23.072,154.048
C09752=1076.067,57.394,434.882,173.581,23.075,154.049
C09753=1076.073,57.644,434.865,173.582,23.077,154.049
C09754=1076.079,57.893,434.849,173.584,23.080,154.049
C09755=1076.085,58.142,434.833,173.585,23.082,154.049
C09756=1076.090,58.392,434.816,173.587,23.085,154.050
C09757=1076.096,58.641,434.800,173.588,23.087,154.050
C09758=1076.103,58.890,434.783,173.590,23.090,154.050
C09759=1076.108,59.139,434.766,173.591,23.092,154.051
C09760=1076.114,59.389,434.750,173.593,23.095,154.051
C09761=1076.120,59.638,434.733,173.594,23.097,154.051
C09762=1076.126,59.888,434.717,173.596,23.100,154.051
C09763=1076.132,60.137,434.700,173.597,23.102,154.052
C09764=1076.138,60.387,434.683,173.599,23.105,154.052
C09765=1076.144,60.636,434.667,173.600,23.107,154.052
C09766=1076.150,60.885,434.650,173.602,23.110,154.053
C09767=1076.155,61.135,434.634,173.603,23.112,154.053
C09768=1076.161,61.384,434.617,173.605,23.115,154.053
C09769=1076.167,61.633,434.600,173.606,23.118,154.053
C09770=1076.173,61.883,434.584,173.608,23.120,154.054
C09771=1076.179,62.132,434.566,173.609,23.122,154.054
C09772=1076.185,62.382,434.550,173.611,23.125,154.054
C09773=1076.192,62.663,434.531,173.612,23.128,154.055
C09774=1076.198,62.944,434.512,173.614,23.130,154.055
C09775=1076.205,63.225,434.494,173.616,23.133,154.055
C09776=1076.212,63.506,434.474,173.618,23.136,154.055
C09777=1076.218,63.755,434.458,173.619,23.139,154.056
C09778=1076.223,64.005,434.441,173.620,23.141,154.056
C09779=1076.229,64.254,434.424,173.622,23.143,154.056
C09780=1076.235,64.503,434.408,173.624,23.146,154.057
C09781=1076.241,64.753,434.391,173.625,23.149,154.057
C09782=1076.247,65.002,434.374,173.626,23.151,154.057
C09783=1076.253,65.252,434.357,173.628,23.153,154.057
C09784=1076.259,65.501,434.341,173.630,23.156,154.058
C09785=1076.264,65.750,434.323,173.631,23.159,154.058
C09786=1076.270,65.999,434.307,173.632,23.161,154.058
C09787=1076.276,66.248,434.289,173.634,23.163,154.059
C09788=1076.281,66.498,434.272,173.636,23.166,154.059
C09789=1076.288,66.748,434.255,173.637,23.169,154.059
C09790=1076.293,66.997,434.238,173.638,23.171,154.059
C09791=1076.299,67.247,434.222,173.640,23.173,154.060
C09792=1076.304,67.496,434.204,173.642,23.176,154.060
C09793=1076.310,67.745,434.188,173.643,23.179,154.060
C09794=1076.316,67.994,434.171,173.644,23.181,154.061
C09795=1076.322,68.244,434.154,173.646,23.183,154.061
C09796=1076.328,68.493,434.136,173.648,23.186,154.061
C09797=1076.334,68.742,434.120,173.649,23.189,154.061
C09798=1076.339,68.991,434.103,173.650,23.191,154.062
C09799=1076.345,69.241,434.086,173.652,23.194,154.062
C09800=1076.351,69.491,434.068,173.654,23.196,154.062
C09801=1076.357,69.740,434.051,173.655,23.199,154.063
C09802=1076.363,69.989,434.035,173.656,23.201,154.063
C09803=1076.368,70.239,434.018,173.658,23.204,154.063
C09804=1076.374,70.488,434.000,173.660,23.206,154.063
C09805=1076.380,70.737,433.983,173.661,23.209,154.064
C09806=1076.386,70.987,433.966,173.662,23.212,154.064
C09807=1076.391,71.236,433.948,173.664,23.214,154.064
C09808=1076.396,71.485,433.931,173.666,23.217,154.065
C09809=1076.403,71.734,433.915,173.667,23.219,154.065
C09810=1076.409,71.984,433.897,173.668,23.222,154.065
C09811=1076.414,72.234,433.880,173.670,23.224,154.065
C09812=1076.420,72.482,433.863,173.672,23.227,154.066
C09813=1076.425,72.732,433.846,173.673,23.229,154.066
C09814=1076.432,72.982,433.828,173.675,23.232,154.066
C09815=1076.437,73.231,433.810,173.676,23.234,154.067
C09816=1076.443,73.480,433.794,173.678,23.237,154.067
C09817=1076.449,73.729,433.777,173.679,23.239,154.067
C09818=1076.455,73.979,433.759,173.681,23.242,154.067
C09819=1076.461,74.228,433.742,173.682,23.244,154.068
C09820=1076.466,74.477,433.725,173.684,23.247,154.068
C09821=1076.472,74.726,433.707,173.685,23.249,154.068
C09822=1076.477,74.977,433.690,173.687,23.252,154.069
C09823=1076.484,75.225,433.673,173.688,23.254,154.069
C09824=1076.489,75.474,433.656,173.690,23.257,154.069
C09825=1076.495,75.723,433.638,173.692,23.260,154.069
C09826=1076.501,75.974,433.621,173.693,23.262,154.070
C09827=1076.506,76.223,433.603,173.694,23.264,154.070
C09828=1076.512,76.472,433.586,173.696,23.267,154.070
C09829=1076.519,76.721,433.568,173.698,23.270,154.071
C09830=1076.524,76.971,433.551,173.699,23.272,154.071
C09831=1076.529,77.220,433.534,173.701,23.274,154.071
C09832=1076.536,77.469,433.516,173.703,23.277,154.071
C09833=1076.542,77.718,433.499,173.704,23.280,154.072
C09834=1076.547,77.968,433.481,173.705,23.282,154.072
C09835=1076.552,78.217,433.465,173.707,23.284,154.072
C09836=1076.558,78.467,433.447,173.709,23.287,154.072
C09837=1076.565,78.747,433.427,173.710,23.290,154.073
C09838=1076.572,79.028,433.407,173.712,23.292,154.073
C09839=1076.578,79.309,433.387,173.713,23.295,154.073
C09840=1076.584,79.591,433.368,173.716,23.298,154.074
C09841=1076.589,79.840,433.350,173.717,23.300,154.074
C09842=1076.595,80.090,433.332,173.719,23.303,154.074
C09843=1076.601,80.339,433.315,173.720,23.306,154.075
C09844=1076.606,80.588,433.297,173.722,23.308,154.075
C09845=1076.613,80.837,433.280,173.724,23.311,154.075
C09846=1076.619,81.086,433.262,173.725,23.313,154.075
C09847=1076.624,81.335,433.245,173.726,23.316,154.076
C09848=1076.631,81.585,433.227,173.728,23.318,154.076
C09849=1076.636,81.834,433.209,173.730,23.321,154.076
C09850=1076.641,82.084,433.192,173.731,23.323,154.077
C09851=1076.647,82.333,433.174,173.732,23.326,154.077
C09852=1076.653,82.582,433.157,173.735,23.328,154.077
C09853=1076.658,82.831,433.139,173.736,23.331,154.077
C09854=1076.665,83.081,433.121,173.737,23.333,154.078
C09855=1076.669,83.331,433.103,173.739,23.336,154.078
C09856=1076.675,83.580,433.086,173.741,23.338,154.078
C09857=1076.681,83.829,433.068,173.742,23.341,154.079
C09858=1076.686,84.078,433.050,173.743,23.343,154.079
C09859=1076.693,84.328,433.032,173.745,23.346,154.079
C09860=1076.698,84.577,433.015,173.747,23.348,154.079
C09861=1076.704,84.826,432.997,173.748,23.351,154.080
C09862=1076.710,85.076,432.979,173.750,23.354,154.080
C09863=1076.716,85.324,432.961,173.751,23.356,154.080
C09864=1076.722,85.574,432.943,173.753,23.358,154.080
C09865=1076.727,85.823,432.925,173.755,23.361,154.081
C09866=1076.733,86.072,432.908,173.756,23.363,154.081
C09867=1076.739,86.322,432.890,173.758,23.366,154.081
C09868=1076.744,86.571,432.872,173.760,23.369,154.082
C09869=1076.750,86.821,432.854,173.761,23.371,154.082
C09870=1076.756,87.070,432.837,173.762,23.373,154.082
C09871=1076.762,87.319,432.819,173.764,23.376,154.082
C09872=1076.768,87.568,432.801,173.766,23.379,154.083
C09873=1076.773,87.817,432.783,173.767,23.380,154.083
C09874=1076.780,88.067,432.765,173.769,23.383,154.083
C09875=1076.785,88.316,432.747,173.771,23.386,154.083
C09876=1076.790,88.566,432.729,173.772,23.388,154.084
C09877=1076.796,88.815,432.711,173.773,23.390,154.084
C09878=1076.802,89.065,432.693,173.776,23.393,154.084
C09879=1076.808,89.313,432.675,173.777,23.396,154.085
C09880=1076.814,89.563,432.657,173.778,23.398,154.085
C09881=1076.820,89.812,432.640,173.780,23.401,154.085
C09882=1076.826,90.061,432.622,173.782,23.403,154.085
C09883=1076.831,90.310,432.604,173.783,23.405,154.086
C09884=1076.838,90.560,432.585,173.785,23.408,154.086
C09885=1076.843,90.809,432.568,173.787,23.410,154.086
C09886=1076.849,91.059,432.549,173.788,23.413,154.086
C09887=1076.854,91.308,432.532,173.790,23.415,154.087
C09888=1076.860,91.557,432.513,173.791,23.418,154.087
C09889=1076.866,91.806,432.496,173.793,23.420,154.087
C09890=1076.871,92.056,432.477,173.795,23.423,154.088
C09891=1076.877,92.304,432.459,173.796,23.425,154.088
C09892=1076.883,92.554,432.441,173.797,23.428,154.088
C09893=1076.888,92.803,432.423,173.800,23.430,154.088
C09894=1076.894,93.053,432.405,173.801,23.433,154.089
C09895=1076.900,93.302,432.386,173.802,23.435,154.089
C09896=1076.905,93.551,432.368,173.804,23.438,154.089
C09897=1076.911,93.801,432.350,173.806,23.440,154.089
C09898=1076.917,94.049,432.332,173.807,23.443,154.090
C09899=1076.922,94.299,432.314,173.809,23.445,154.090
C09900=1076.928,94.548,432.295,173.811,23.447,154.090
C09901=1076.935,94.829,432.275,173.813,23.451,154.091
C09902=1076.941,95.110,432.255,173.814,23.453,154.091
C09903=1076.947,95.391,432.233,173.816,23.456,154.091
C09904=1076.954,95.672,432.213,173.818,23.459,154.092
C09905=1076.960,95.922,432.195,173.820,23.461,154.092
C09906=1076.966,96.170,432.177,173.821,23.463,154.092
C09907=1076.971,96.420,432.158,173.823,23.466,154.092
C09908=1076.977,96.669,432.140,173.825,23.469,154.093
C09909=1076.983,96.919,432.122,173.826,23.471,154.093
C09910=1076.988,97.167,432.103,173.828,23.474,154.093
C09911=1076.994,97.417,432.085,173.829,23.476,154.093
C09912=1077.000,97.667,432.066,173.831,23.479,154.094
C09913=1077.005,97.916,432.049,173.833,23.481,154.094
C09914=1077.012,98.165,432.030,173.834,23.483,154.094
C09915=1077.017,98.414,432.012,173.836,23.486,154.094
C09916=1077.023,98.663,431.993,173.838,23.488,154.095
C09917=1077.029,98.912,431.975,173.839,23.491,154.095
C09918=1077.034,99.162,431.956,173.841,23.493,154.095
C09919=1077.040,99.411,431.938,173.843,23.496,154.095
C09920=1077.045,99.660,431.919,173.844,23.498,154.096
C09921=1077.052,99.910,431.902,173.846,23.500,154.096
C09922=1077.058,100.159,431.883,173.848,23.503,154.096
C09923=1077.063,100.408,431.865,173.849,23.505,154.097
C09924=1077.069,100.657,431.846,173.851,23.508,154.097
C09925=1077.074,100.906,431.827,173.852,23.510,154.097
C09926=1077.080,101.156,431.809,173.854,23.512,154.097
C09927=1077.086,101.405,431.790,173.856,23.515,154.097
C09928=1077.092,101.654,431.772,173.857,23.517,154.098
C09929=1077.097,101.904,431.753,173.860,23.520,154.098
C09930=1077.103,102.152,431.735,173.861,23.523,154.098
C09931=1077.108,102.402,431.716,173.862,23.525,154.099
C09932=1077.114,102.652,431.697,173.864,23.528,154.099
C09933=1077.120,102.900,431.679,173.866,23.530,154.099
C09934=1077.125,103.150,431.660,173.867,23.532,154.099
C09935=1077.132,103.399,431.642,173.869,23.535,154.100
C09936=1077.137,103.648,431.623,173.871,23.537,154.100
C09937=1077.142,103.898,431.604,173.872,23.539,154.100
C09938=1077.148,104.147,431.586,173.874,23.542,154.100
C09939=1077.154,104.396,431.567,173.876,23.545,154.101
C09940=1077.160,104.645,431.548,173.878,23.547,154.101
C09941=1077.165,104.894,431.530,173.879,23.550,154.101
C09942=1077.171,105.144,431.511,173.880,23.552,154.102
C09943=1077.177,105.393,431.492,173.883,23.555,154.102
C09944=1077.182,105.642,431.474,173.884,23.557,154.102
C09945=1077.188,105.892,431.455,173.886,23.560,154.102
C09946=1077.194,106.141,431.436,173.888,23.562,154.103
C09947=1077.199,106.390,431.417,173.889,23.564,154.103
C09948=1077.206,106.639,431.398,173.891,23.567,154.103
C09949=1077.211,106.889,431.380,173.892,23.569,154.103
C09950=1077.216,107.138,431.361,173.894,23.571,154.104
C09951=1077.222,107.387,431.342,173.896,23.574,154.104
C09952=1077.228,107.636,431.323,173.897,23.576,154.104
C09953=1077.234,107.886,431.304,173.900,23.579,154.104
C09954=1077.240,108.134,431.286,173.901,23.582,154.105
C09955=1077.245,108.384,431.267,173.902,23.583,154.105
C09956=1077.251,108.633,431.248,173.905,23.586,154.105
C09957=1077.256,108.882,431.230,173.906,23.589,154.105
C09958=1077.262,109.131,431.210,173.908,23.591,154.106
C09959=1077.268,109.381,431.191,173.909,23.594,154.106
C09960=1077.274,109.630,431.172,173.911,23.596,154.106
C09961=1077.279,109.879,431.154,173.913,23.598,154.106
C09962=1077.285,110.128,431.134,173.914,23.601,154.107
C09963=1077.291,110.377,431.116,173.917,23.603,154.107
C09964=1077.297,110.627,431.096,173.918,23.605,154.107
C09965=1077.303,110.908,431.075,173.920,23.609,154.107
C09966=1077.310,111.189,431.055,173.921,23.611,154.108
C09967=1077.316,111.470,431.033,173.924,23.614,154.108
C09968=1077.323,111.751,431.011,173.926,23.616,154.108
C09969=1077.328,112.001,430.992,173.927,23.619,154.109
C09970=1077.334,112.249,430.974,173.929,23.622,154.109
C09971=1077.340,112.499,430.954,173.931,23.623,154.109
C09972=1077.345,112.748,430.935,173.933,23.626,154.109
C09973=1077.351,112.997,430.916,173.934,23.629,154.110
C09974=1077.356,113.246,430.897,173.936,23.631,154.110
C09975=1077.362,113.496,430.878,173.938,23.634,154.110
C09976=1077.368,113.745,430.859,173.939,23.636,154.110
C09977=1077.374,113.994,430.840,173.942,23.638,154.111
C09978=1077.380,114.244,430.821,173.943,23.641,154.111
C09979=1077.385,114.492,430.801,173.944,23.643,154.111
C09980=1077.391,114.741,430.782,173.947,23.645,154.111
C09981=1077.397,114.991,430.763,173.948,23.648,154.112
C09982=1077.402,115.240,430.743,173.950,23.650,154.112
C09983=1077.407,115.489,430.725,173.951,23.653,154.112
C09984=1077.413,115.738,430.705,173.954,23.656,154.112
C09985=1077.419,115.988,430.686,173.955,23.658,154.113
C09986=1077.424,116.237,430.667,173.956,23.660,154.113
C09987=1077.429,116.486,430.648,173.959,23.663,154.113
C09988=1077.435,116.735,430.628,173.960,23.665,154.113
C09989=1077.441,116.984,430.609,173.962,23.668,154.114
C09990=1077.447,117.233,430.590,173.964,23.670,154.114
C09991=1077.453,117.483,430.570,173.966,23.673,154.114
C09992=1077.458,117.732,430.551,173.967,23.675,154.114
C09993=1077.464,117.980,430.531,173.969,23.677,154.115
C09994=1077.469,118.230,430.512,173.971,23.680,154.115
C09995=1077.474,118.480,430.492,173.972,23.682,154.115
C09996=1077.480,118.729,430.473,173.974,23.685,154.115
//INST
///DATE 2021/06/25 14:45
///ATTR SC,RW,RJ
////FRAME ROBOT
///GROUP1 RB1
NOP
MOVL C00000 V=800.0 PL=0
MOVL C00001 V=800.0 PL=0
MOVL C00002 V=800.0 PL=0
MOVL C00003 V=800.0 PL=0
MOVL C00004 V=800.0 PL=0
MOVL C00005 V=800.0 PL=0
MOVL C00006 V=800.0 PL=0
MOVL C00007 V=800.0 PL=0
MOVL C00008 V=800.0 PL=0
MOVL C00009 V=800.0 PL=0
MOVL C00010 V=800.0 PL=0
MOVL C00011 V=800.0 PL=0
MOVL C00012 V=800.0 PL=0
MOVL C00013 V=800.0 PL=0
MOVL C00014 V=800.0 PL=0
MOVL C00015 V=800.0 PL=0
MOVL C00016 V=800.0 PL=0
MOVL C00017 V=800.0 PL=0
MOVL C00018 V=800.0 PL=0
MOVL C00019 V=800.0 PL=0
MOVL C00020 V=800.0 PL=0
MOVL C00021 V=800.0 PL=0
MOVL C00022 V=800.0 PL=0
MOVL C00023 V=800.0 PL=0
MOVL C00024 V=800.0 PL=0
MOVL C00025 V=800.0 PL=0
MOVL C00026 V=800.0 PL=0
MOVL C00027 V=800.0 PL=0
MOVL C00028 V=800.0 PL=0
MOVL C00029 V=800.0 PL=0
MOVL C00030 V=800.0 PL=0
MOVL C00031 V=800.0 PL=0
MOVL C00032 V=800.0 PL=0
MOVL C00033 V=800.0 PL=0
MOVL C00034 V=800.0 PL=0
MOVL C00035 V=800.0 PL=0
MOVL C00036 V=800.0 PL=0
MOVL C00037 V=800.0 PL=0
MOVL C00038 V=800.0 PL=0
MOVL C00039 V=800.0 PL=0
MOVL C00040 V=800.0 PL=0
MOVL C00041 V=800.0 PL=0
MOVL C00042 V=800.0 PL=0
MOVL C00043 V=800.0 PL=0
MOVL C00044 V=800.0 PL=0
MOVL C00045 V=800.0 PL=0
MOVL C00046 V=800.0 PL=0
MOVL C00047 V=800.0 PL=0
MOVL C00048 V=800.0 PL=0
MOVL C00049 V=800.0 PL=0
MOVL C00050 V=800.0 PL=0
MOVL C00051 V=800.0 PL=0
MOVL C00052 V=800.0 PL=0
MOVL C00053 V=800.0 PL=0
MOVL C00054 V=800.0 PL=0
MOVL C00055 V=800.0 PL=0
MOVL C00056 V=800.0 PL=0
MOVL C00057 V=800.0 PL=0
MOVL C00058 V=800.0 PL=0
MOVL C00059 V=800.0 PL=0
MOVL C00060 V=800.0 PL=0
MOVL C00061 V=800.0 PL=0
MOVL C00062 V=800.0 PL=0
MOVL C00063 V=800.0 PL=0
MOVL C00064 V=800.0 PL=0
MOVL C00065 V=800.0 PL=0
MOVL C00066 V=800.0 PL=0
MOVL C00067 V=800.0 PL=0
MOVL C00068 V=800.0 PL=0
MOVL C00069 V=800.0 PL=0
MOVL C00070 V=800.0 PL=0
MOVL C00071 V=800.0 PL=0
MOVL C00072 V=800.0 PL=0
MOVL C00073 V=800.0 PL=0
MOVL C00074 V=800.0 PL=0
MOVL C00075 V=800.0 PL=0
MOVL C00076 V=800.0 PL=0
MOVL C00077 V=800.0 PL=0
MOVL C00078 V=800.0 PL=0
MOVL C00079 V=800.0 PL=0
MOVL C00080 V=800.0 PL=0
MOVL C00081 V=800.0 PL=0
MOVL C00082 V=800.0 PL=0
MOVL C00083 V=800.0 PL=0
MOVL C00084 V=800.0 PL=0
MOVL C00085 V=800.0 PL=0
MOVL C00086 V=800.0 PL=0
MOVL C00087 V=800.0 PL=0
MOVL C00088 V=800.0 PL=0
MOVL C00089 V=800.0 PL=0
MOVL C00090 V=800.0 PL=0
MOVL C00091 V=800.0 PL=0
MOVL C00092 V=800.0 PL=0
MOVL C00093 V=800.0 PL=0
MOVL C00094 V=800.0 PL=0
MOVL C00095 V=800.0 PL=0
MOVL C00096 V=800.0 PL=0
MOVL C00097 V=800.0 PL=0
MOVL C00098 V=800.0 PL=0
MOVL C00099 V=800.0 PL=0
MOVL C00100 V=800.0 PL=0
MOVL C00101 V=800.0 PL=0
MOVL C00102 V=800.0 PL=0
MOVL C00103 V=800.0 PL=0
MOVL C00104 V=800.0 PL=0
MOVL C00105 V=800.0 PL=0
MOVL C00106 V=800.0 PL=0
MOVL C00107 V=800.0 PL=0
MOVL C00108 V=800.0 PL=0
MOVL C00109 V=800.0 PL=0
MOVL C00110 V=800.0 PL=0
MOVL C00111 V=800.0 PL=0
MOVL C00112 V=800.0 PL=0
MOVL C00113 V=800.0 PL=0
MOVL C00114 V=800.0 PL=0
MOVL C00115 V=800.0 PL=0
MOVL C00116 V=800.0 PL=0
MOVL C00117 V=800.0 PL=0
MOVL C00118 V=800.0 PL=0
MOVL C00119 V=800.0 PL=0
MOVL C00120 V=800.0 PL=0
MOVL C00121 V=800.0 PL=0
MOVL C00122 V=800.0 PL=0
MOVL C00123 V=800.0 PL=0
MOVL C00124 V=800.0 PL=0
MOVL C00125 V=800.0 PL=0
MOVL C00126 V=800.0 PL=0
MOVL C00127 V=800.0 PL=0
MOVL C00128 V=800.0 PL=0
MOVL C00129 V=800.0 PL=0
MOVL C00130 V=800.0 PL=0
MOVL C00131 V=800.0 PL=0
MOVL C00132 V=800.0 PL=0
MOVL C00133 V=800.0 PL=0
MOVL C00134 V=800.0 PL=0
MOVL C00135 V=800.0 PL=0
MOVL C00136 V=800.0 PL=0
MOVL C00137 V=800.0 PL=0
MOVL C00138 V=800.0 PL=0
MOVL C00139 V=800.0 PL=0
MOVL C00140 V=800.0 PL=0
MOVL C00141 V=800.0 PL=0
MOVL C00142 V=800.0 PL=0
MOVL C00143 V=800.0 PL=0
MOVL C00144 V=800.0 PL=0
MOVL C00145 V=800.0 PL=0
MOVL C00146 V=800.0 PL=0
MOVL C00147 V=800.0 PL=0
MOVL C00148 V=800.0 PL=0
MOVL C00149 V=800.0 PL=0
MOVL C00150 V=800.0 PL=0
MOVL C00151 V=800.0 PL=0
MOVL C00152 V=800.0 PL=0
MOVL C00153 V=800.0 PL=0
MOVL C00154 V=800.0 PL=0
MOVL C00155 V=800.0 PL=0
MOVL C00156 V=800.0 PL=0
MOVL C00157 V=800.0 PL=0
MOVL C00158 V=800.0 PL=0
MOVL C00159 V=800.0 PL=0
MOVL C00160 V=800.0 PL=0
MOVL C00161 V=800.0 PL=0
MOVL C00162 V=800.0 PL=0
MOVL C00163 V=800.0 PL=0
MOVL C00164 V=800.0 PL=0
MOVL C00165 V=800.0 PL=0
MOVL C00166 V=800.0 PL=0
MOVL C00167 V=800.0 PL=0
MOVL C00168 V=800.0 PL=0
MOVL C00169 V=800.0 PL=0
MOVL C00170 V=800.0 PL=0
MOVL C00171 V=800.0 PL=0
MOVL C00172 V=800.0 PL=0
MOVL C00173 V=800.0 PL=0
MOVL C00174 V=800.0 PL=0
MOVL C00175 V=800.0 PL=0
MOVL C00176 V=800.0 PL=0
MOVL C00177 V=800.0 PL=0
MOVL C00178 V=800.0 PL=0
MOVL C00179 V=800.0 PL=0
MOVL C00180 V=800.0 PL=0
MOVL C00181 V=800.0 PL=0
MOVL C00182 V=800.0 PL=0
MOVL C00183 V=800.0 PL=0
MOVL C00184 V=800.0 PL=0
MOVL C00185 V=800.0 PL=0
MOVL C00186 V=800.0 PL=0
MOVL C00187 V=800.0 PL=0
MOVL C00188 V=800.0 PL=0
MOVL C00189 V=800.0 PL=0
MOVL C00190 V=800.0 PL=0
MOVL C00191 V=800.0 PL=0
MOVL C00192 V=800.0 PL=0
MOVL C00193 V=800.0 PL=0
MOVL C00194 V=800.0 PL=0
MOVL C00195 V=800.0 PL=0
MOVL C00196 V=800.0 PL=0
MOVL C00197 V=800.0 PL=0
MOVL C00198 V=800.0 PL=0
MOVL C00199 V=800.0 PL=0
MOVL C00200 V=800.0 PL=0
MOVL C00201 V=800.0 PL=0
MOVL C00202 V=800.0 PL=0
MOVL C00203 V=800.0 PL=0
MOVL C00204 V=800.0 PL=0
MOVL C00205 V=800.0 PL=0
MOVL C00206 V=800.0 PL=0
MOVL C00207 V=800.0 PL=0
MOVL C00208 V=800.0 PL=0
MOVL C00209 V=800.0 PL=0
MOVL C00210 V=800.0 PL=0
MOVL C00211 V=800.0 PL=0
MOVL C00212 V=800.0 PL=0
MOVL C00213 V=800.0 PL=0
MOVL C00214 V=800.0 PL=0
MOVL C00215 V=800.0 PL=0
MOVL C00216 V=800.0 PL=0
MOVL C00217 V=800.0 PL=0
MOVL C00218 V=800.0 PL=0
MOVL C00219 V=800.0 PL=0
MOVL C00220 V=800.0 PL=0
MOVL C00221 V=800.0 PL=0
MOVL C00222 V=800.0 PL=0
MOVL C00223 V=800.0 PL=0
MOVL C00224 V=800.0 PL=0
MOVL C00225 V=800.0 PL=0
MOVL C00226 V=800.0 PL=0
MOVL C00227 V=800.0 PL=0
MOVL C00228 V=800.0 PL=0
MOVL C00229 V=800.0 PL=0
MOVL C00230 V=800.0 PL=0
MOVL C00231 V=800.0 PL=0
MOVL C00232 V=800.0 PL=0
MOVL C00233 V=800.0 PL=0
MOVL C00234 V=800.0 PL=0
MOVL C00235 V=800.0 PL=0
MOVL C00236 V=800.0 PL=0
MOVL C00237 V=800.0 PL=0
MOVL C00238 V=800.0 PL=0
MOVL C00239 V=800.0 PL=0
MOVL C00240 V=800.0 PL=0
MOVL C00241 V=800.0 PL=0
MOVL C00242 V=800.0 PL=0
MOVL C00243 V=800.0 PL=0
MOVL C00244 V=800.0 PL=0
MOVL C00245 V=800.0 PL=0
MOVL C00246 V=800.0 PL=0
MOVL C00247 V=800.0 PL=0
MOVL C00248 V=800.0 PL=0
MOVL C00249 V=800.0 PL=0
MOVL C00250 V=800.0 PL=0
MOVL C00251 V=800.0 PL=0
MOVL C00252 V=800.0 PL=0
MOVL C00253 V=800.0 PL=0
MOVL C00254 V=800.0 PL=0
MOVL C00255 V=800.0 PL=0
MOVL C00256 V=800.0 PL=0
MOVL C00257 V=800.0 PL=0
MOVL C00258 V=800.0 PL=0
MOVL C00259 V=800.0 PL=0
MOVL C00260 V=800.0 PL=0
MOVL C00261 V=800.0 PL=0
MOVL C00262 V=800.0 PL=0
MOVL C00263 V=800.0 PL=0
MOVL C00264 V=800.0 PL=0
MOVL C00265 V=800.0 PL=0
MOVL C00266 V=800.0 PL=0
MOVL C00267 V=800.0 PL=0
MOVL C00268 V=800.0 PL=0
MOVL C00269 V=800.0 PL=0
MOVL C00270 V=800.0 PL=0
MOVL C00271 V=800.0 PL=0
MOVL C00272 V=800.0 PL=0
MOVL C00273 V=800.0 PL=0
MOVL C00274 V=800.0 PL=0
MOVL C00275 V=800.0 PL=0
MOVL C00276 V=800.0 PL=0
MOVL C00277 V=800.0 PL=0
MOVL C00278 V=800.0 PL=0
MOVL C00279 V=800.0 PL=0
MOVL C00280 V=800.0 PL=0
MOVL C00281 V=800.0 PL=0
MOVL C00282 V=800.0 PL=0
MOVL C00283 V=800.0 PL=0
MOVL C00284 V=800.0 PL=0
MOVL C00285 V=800.0 PL=0
MOVL C00286 V=800.0 PL=0
MOVL C00287 V=800.0 PL=0
MOVL C00288 V=800.0 PL=0
MOVL C00289 V=800.0 PL=0
MOVL C00290 V=800.0 PL=0
MOVL C00291 V=800.0 PL=0
MOVL C00292 V=800.0 PL=0
MOVL C00293 V=800.0 PL=0
MOVL C00294 V=800.0 PL=0
MOVL C00295 V=800.0 PL=0
MOVL C00296 V=800.0 PL=0
MOVL C00297 V=800.0 PL=0
MOVL C00298 V=800.0 PL=0
MOVL C00299 V=800.0 PL=0
MOVL C00300 V=800.0 PL=0
MOVL C00301 V=800.0 PL=0
MOVL C00302 V=800.0 PL=0
MOVL C00303 V=800.0 PL=0
MOVL C00304 V=800.0 PL=0
MOVL C00305 V=800.0 PL=0
MOVL C00306 V=800.0 PL=0
MOVL C00307 V=800.0 PL=0
MOVL C00308 V=800.0 PL=0
MOVL C00309 V=800.0 PL=0
MOVL C00310 V=800.0 PL=0
MOVL C00311 V=800.0 PL=0
MOVL C00312 V=800.0 PL=0
MOVL C00313 V=800.0 PL=0
MOVL C00314 V=800.0 PL=0
MOVL C00315 V=800.0 PL=0
MOVL C00316 V=800.0 PL=0
MOVL C00317 V=800.0 PL=0
MOVL C00318 V=800.0 PL=0
MOVL C00319 V=800.0 PL=0
MOVL C00320 V=800.0 PL=0
MOVL C00321 V=800.0 PL=0
MOVL C00322 V=800.0 PL=0
MOVL C00323 V=800.0 PL=0
MOVL C00324 V=800.0 PL=0
MOVL C00325 V=800.0 PL=0
MOVL C00326 V=800.0 PL=0
MOVL C00327 V=800.0 PL=0
MOVL C00328 V=800.0 PL=0
MOVL C00329 V=800.0 PL=0
MOVL C00330 V=800.0 PL=0
MOVL C00331 V=800.0 PL=0
MOVL C00332 V=800.0 PL=0
MOVL C00333 V=800.0 PL=0
MOVL C00334 V=800.0 PL=0
MOVL C00335 V=800.0 PL=0
MOVL C00336 V=800.0 PL=0
MOVL C00337 V=800.0 PL=0
MOVL C00338 V=800.0 PL=0
MOVL C00339 V=800.0 PL=0
MOVL C00340 V=800.0 PL=0
MOVL C00341 V=800.0 PL=0
MOVL C00342 V=800.0 PL=0
MOVL C00343 V=800.0 PL=0
MOVL C00344 V=800.0 PL=0
MOVL C00345 V=800.0 PL=0
MOVL C00346 V=800.0 PL=0
MOVL C00347 V=800.0 PL=0
MOVL C00348 V=800.0 PL=0
MOVL C00349 V=800.0 PL=0
MOVL C00350 V=800.0 PL=0
MOVL C00351 V=800.0 PL=0
MOVL C00352 V=800.0 PL=0
MOVL C00353 V=800.0 PL=0
MOVL C00354 V=800.0 PL=0
MOVL C00355 V=800.0 PL=0
MOVL C00356 V=800.0 PL=0
MOVL C00357 V=800.0 PL=0
MOVL C00358 V=800.0 PL=0
MOVL C00359 V=800.0 PL=0
MOVL C00360 V=800.0 PL=0
MOVL C00361 V=800.0 PL=0
MOVL C00362 V=800.0 PL=0
MOVL C00363 V=800.0 PL=0
MOVL C00364 V=800.0 PL=0
MOVL C00365 V=800.0 PL=0
MOVL C00366 V=800.0 PL=0
MOVL C00367 V=800.0 PL=0
MOVL C00368 V=800.0 PL=0
MOVL C00369 V=800.0 PL=0
MOVL C00370 V=800.0 PL=0
MOVL C00371 V=800.0 PL=0
MOVL C00372 V=800.0 PL=0
MOVL C00373 V=800.0 PL=0
MOVL C00374 V=800.0 PL=0
MOVL C00375 V=800.0 PL=0
MOVL C00376 V=800.0 PL=0
MOVL C00377 V=800.0 PL=0
MOVL C00378 V=800.0 PL=0
MOVL C00379 V=800.0 PL=0
MOVL C00380 V=800.0 PL=0
MOVL C00381 V=800.0 PL=0
MOVL C00382 V=800.0 PL=0
MOVL C00383 V=800.0 PL=0
MOVL C00384 V=800.0 PL=0
MOVL C00385 V=800.0 PL=0
MOVL C00386 V=800.0 PL=0
MOVL C00387 V=800.0 PL=0
MOVL C00388 V=800.0 PL=0
MOVL C00389 V=800.0 PL=0
MOVL C00390 V=800.0 PL=0
MOVL C00391 V=800.0 PL=0
MOVL C00392 V=800.0 PL=0
MOVL C00393 V=800.0 PL=0
MOVL C00394 V=800.0 PL=0
MOVL C00395 V=800.0 PL=0
MOVL C00396 V=800.0 PL=0
MOVL C00397 V=800.0 PL=0
MOVL C00398 V=800.0 PL=0
MOVL C00399 V=800.0 PL=0
MOVL C00400 V=800.0 PL=0
MOVL C00401 V=800.0 PL=0
MOVL C00402 V=800.0 PL=0
MOVL C00403 V=800.0 PL=0
MOVL C00404 V=800.0 PL=0
MOVL C00405 V=800.0 PL=0
MOVL C00406 V=800.0 PL=0
MOVL C00407 V=800.0 PL=0
MOVL C00408 V=800.0 PL=0
MOVL C00409 V=800.0 PL=0
MOVL C00410 V=800.0 PL=0
MOVL C00411 V=800.0 PL=0
MOVL C00412 V=800.0 PL=0
MOVL C00413 V=800.0 PL=0
MOVL C00414 V=800.0 PL=0
MOVL C00415 V=800.0 PL=0
MOVL C00416 V=800.0 PL=0
MOVL C00417 V=800.0 PL=0
MOVL C00418 V=800.0 PL=0
MOVL C00419 V=800.0 PL=0
MOVL C00420 V=800.0 PL=0
MOVL C00421 V=800.0 PL=0
MOVL C00422 V=800.0 PL=0
MOVL C00423 V=800.0 PL=0
MOVL C00424 V=800.0 PL=0
MOVL C00425 V=800.0 PL=0
MOVL C00426 V=800.0 PL=0
MOVL C00427 V=800.0 PL=0
MOVL C00428 V=800.0 PL=0
MOVL C00429 V=800.0 PL=0
MOVL C00430 V=800.0 PL=0
MOVL C00431 V=800.0 PL=0
MOVL C00432 V=800.0 PL=0
MOVL C00433 V=800.0 PL=0
MOVL C00434 V=800.0 PL=0
MOVL C00435 V=800.0 PL=0
MOVL C00436 V=800.0 PL=0
MOVL C00437 V=800.0 PL=0
MOVL C00438 V=800.0 PL=0
MOVL C00439 V=800.0 PL=0
MOVL C00440 V=800.0 PL=0
MOVL C00441 V=800.0 PL=0
MOVL C00442 V=800.0 PL=0
MOVL C00443 V=800.0 PL=0
MOVL C00444 V=800.0 PL=0
MOVL C00445 V=800.0 PL=0
MOVL C00446 V=800.0 PL=0
MOVL C00447 V=800.0 PL=0
MOVL C00448 V=800.0 PL=0
MOVL C00449 V=800.0 PL=0
MOVL C00450 V=800.0 PL=0
MOVL C00451 V=800.0 PL=0
MOVL C00452 V=800.0 PL=0
MOVL C00453 V=800.0 PL=0
MOVL C00454 V=800.0 PL=0
MOVL C00455 V=800.0 PL=0
MOVL C00456 V=800.0 PL=0
MOVL C00457 V=800.0 PL=0
MOVL C00458 V=800.0 PL=0
MOVL C00459 V=800.0 PL=0
MOVL C00460 V=800.0 PL=0
MOVL C00461 V=800.0 PL=0
MOVL C00462 V=800.0 PL=0
MOVL C00463 V=800.0 PL=0
MOVL C00464 V=800.0 PL=0
MOVL C00465 V=800.0 PL=0
MOVL C00466 V=800.0 PL=0
MOVL C00467 V=800.0 PL=0
MOVL C00468 V=800.0 PL=0
MOVL C00469 V=800.0 PL=0
MOVL C00470 V=800.0 PL=0
MOVL C00471 V=800.0 PL=0
MOVL C00472 V=800.0 PL=0
MOVL C00473 V=800.0 PL=0
MOVL C00474 V=800.0 PL=0
MOVL C00475 V=800.0 PL=0
MOVL C00476 V=800.0 PL=0
MOVL C00477 V=800.0 PL=0
MOVL C00478 V=800.0 PL=0
MOVL C00479 V=800.0 PL=0
MOVL C00480 V=800.0 PL=0
MOVL C00481 V=800.0 PL=0
MOVL C00482 V=800.0 PL=0
MOVL C00483 V=800.0 PL=0
MOVL C00484 V=800.0 PL=0
MOVL C00485 V=800.0 PL=0
MOVL C00486 V=800.0 PL=0
MOVL C00487 V=800.0 PL=0
MOVL C00488 V=800.0 PL=0
MOVL C00489 V=800.0 PL=0
MOVL C00490 V=800.0 PL=0
MOVL C00491 V=800.0 PL=0
MOVL C00492 V=800.0 PL=0
MOVL C00493 V=800.0 PL=0
MOVL C00494 V=800.0 PL=0
MOVL C00495 V=800.0 PL=0
MOVL C00496 V=800.0 PL=0
MOVL C00497 V=800.0 PL=0
MOVL C00498 V=800.0 PL=0
MOVL C00499 V=800.0 PL=0
MOVL C00500 V=800.0 PL=0
MOVL C00501 V=800.0 PL=0
MOVL C00502 V=800.0 PL=0
MOVL C00503 V=800.0 PL=0
MOVL C00504 V=800.0 PL=0
MOVL C00505 V=800.0 PL=0
MOVL C00506 V=800.0 PL=0
MOVL C00507 V=800.0 PL=0
MOVL C00508 V=800.0 PL=0
MOVL C00509 V=800.0 PL=0
MOVL C00510 V=800.0 PL=0
MOVL C00511 V=800.0 PL=0
MOVL C00512 V=800.0 PL=0
MOVL C00513 V=800.0 PL=0
MOVL C00514 V=800.0 PL=0
MOVL C00515 V=800.0 PL=0
MOVL C00516 V=800.0 PL=0
MOVL C00517 V=800.0 PL=0
MOVL C00518 V=800.0 PL=0
MOVL C00519 V=800.0 PL=0
MOVL C00520 V=800.0 PL=0
MOVL C00521 V=800.0 PL=0
MOVL C00522 V=800.0 PL=0
MOVL C00523 V=800.0 PL=0
MOVL C00524 V=800.0 PL=0
MOVL C00525 V=800.0 PL=0
MOVL C00526 V=800.0 PL=0
MOVL C00527 V=800.0 PL=0
MOVL C00528 V=800.0 PL=0
MOVL C00529 V=800.0 PL=0
MOVL C00530 V=800.0 PL=0
MOVL C00531 V=800.0 PL=0
MOVL C00532 V=800.0 PL=0
MOVL C00533 V=800.0 PL=0
MOVL C00534 V=800.0 PL=0
MOVL C00535 V=800.0 PL=0
MOVL C00536 V=800.0 PL=0
MOVL C00537 V=800.0 PL=0
MOVL C00538 V=800.0 PL=0
MOVL C00539 V=800.0 PL=0
MOVL C00540 V=800.0 PL=0
MOVL C00541 V=800.0 PL=0
MOVL C00542 V=800.0 PL=0
MOVL C00543 V=800.0 PL=0
MOVL C00544 V=800.0 PL=0
MOVL C00545 V=800.0 PL=0
MOVL C00546 V=800.0 PL=0
MOVL C00547 V=800.0 PL=0
MOVL C00548 V=800.0 PL=0
MOVL C00549 V=800.0 PL=0
MOVL C00550 V=800.0 PL=0
MOVL C00551 V=800.0 PL=0
MOVL C00552 V=800.0 PL=0
MOVL C00553 V=800.0 PL=0
MOVL C00554 V=800.0 PL=0
MOVL C00555 V=800.0 PL=0
MOVL C00556 V=800.0 PL=0
MOVL C00557 V=800.0 PL=0
MOVL C00558 V=800.0 PL=0
MOVL C00559 V=800.0 PL=0
MOVL C00560 V=800.0 PL=0
MOVL C00561 V=800.0 PL=0
MOVL C00562 V=800.0 PL=0
MOVL C00563 V=800.0 PL=0
MOVL C00564 V=800.0 PL=0
MOVL C00565 V=800.0 PL=0
MOVL C00566 V=800.0 PL=0
MOVL C00567 V=800.0 PL=0
MOVL C00568 V=800.0 PL=0
MOVL C00569 V=800.0 PL=0
MOVL C00570 V=800.0 PL=0
MOVL C00571 V=800.0 PL=0
MOVL C00572 V=800.0 PL=0
MOVL C00573 V=800.0 PL=0
MOVL C00574 V=800.0 PL=0
MOVL C00575 V=800.0 PL=0
MOVL C00576 V=800.0 PL=0
MOVL C00577 V=800.0 PL=0
MOVL C00578 V=800.0 PL=0
MOVL C00579 V=800.0 PL=0
MOVL C00580 V=800.0 PL=0
MOVL C00581 V=800.0 PL=0
MOVL C00582 V=800.0 PL=0
MOVL C00583 V=800.0 PL=0
MOVL C00584 V=800.0 PL=0
MOVL C00585 V=800.0 PL=0
MOVL C00586 V=800.0 PL=0
MOVL C00587 V=800.0 PL=0
MOVL C00588 V=800.0 PL=0
MOVL C00589 V=800.0 PL=0
MOVL C00590 V=800.0 PL=0
MOVL C00591 V=800.0 PL=0
MOVL C00592 V=800.0 PL=0
MOVL C00593 V=800.0 PL=0
MOVL C00594 V=800.0 PL=0
MOVL C00595 V=800.0 PL=0
MOVL C00596 V=800.0 PL=0
MOVL C00597 V=800.0 PL=0
MOVL C00598 V=800.0 PL=0
MOVL C00599 V=800.0 PL=0
MOVL C00600 V=800.0 PL=0
MOVL C00601 V=800.0 PL=0
MOVL C00602 V=800.0 PL=0
MOVL C00603 V=800.0 PL=0
MOVL C00604 V=800.0 PL=0
MOVL C00605 V=800.0 PL=0
MOVL C00606 V=800.0 PL=0
MOVL C00607 V=800.0 PL=0
MOVL C00608 V=800.0 PL=0
MOVL C00609 V=800.0 PL=0
MOVL C00610 V=800.0 PL=0
MOVL C00611 V=800.0 PL=0
MOVL C00612 V=800.0 PL=0
MOVL C00613 V=800.0 PL=0
MOVL C00614 V=800.0 PL=0
MOVL C00615 V=800.0 PL=0
MOVL C00616 V=800.0 PL=0
MOVL C00617 V=800.0 PL=0
MOVL C00618 V=800.0 PL=0
MOVL C00619 V=800.0 PL=0
MOVL C00620 V=800.0 PL=0
MOVL C00621 V=800.0 PL=0
MOVL C00622 V=800.0 PL=0
MOVL C00623 V=800.0 PL=0
MOVL C00624 V=800.0 PL=0
MOVL C00625 V=800.0 PL=0
MOVL C00626 V=800.0 PL=0
MOVL C00627 V=800.0 PL=0
MOVL C00628 V=800.0 PL=0
MOVL C00629 V=800.0 PL=0
MOVL C00630 V=800.0 PL=0
MOVL C00631 V=800.0 PL=0
MOVL C00632 V=800.0 PL=0
MOVL C00633 V=800.0 PL=0
MOVL C00634 V=800.0 PL=0
MOVL C00635 V=800.0 PL=0
MOVL C00636 V=800.0 PL=0
MOVL C00637 V=800.0 PL=0
MOVL C00638 V=800.0 PL=0
MOVL C00639 V=800.0 PL=0
MOVL C00640 V=800.0 PL=0
MOVL C00641 V=800.0 PL=0
MOVL C00642 V=800.0 PL=0
MOVL C00643 V=800.0 PL=0
MOVL C00644 V=800.0 PL=0
MOVL C00645 V=800.0 PL=0
MOVL C00646 V=800.0 PL=0
MOVL C00647 V=800.0 PL=0
MOVL C00648 V=800.0 PL=0
MOVL C00649 V=800.0 PL=0
MOVL C00650 V=800.0 PL=0
MOVL C00651 V=800.0 PL=0
MOVL C00652 V=800.0 PL=0
MOVL C00653 V=800.0 PL=0
MOVL C00654 V=800.0 PL=0
MOVL C00655 V=800.0 PL=0
MOVL C00656 V=800.0 PL=0
MOVL C00657 V=800.0 PL=0
MOVL C00658 V=800.0 PL=0
MOVL C00659 V=800.0 PL=0
MOVL C00660 V=800.0 PL=0
MOVL C00661 V=800.0 PL=0
MOVL C00662 V=800.0 PL=0
MOVL C00663 V=800.0 PL=0
MOVL C00664 V=800.0 PL=0
MOVL C00665 V=800.0 PL=0
MOVL C00666 V=800.0 PL=0
MOVL C00667 V=800.0 PL=0
MOVL C00668 V=800.0 PL=0
MOVL C00669 V=800.0 PL=0
MOVL C00670 V=800.0 PL=0
MOVL C00671 V=800.0 PL=0
MOVL C00672 V=800.0 PL=0
MOVL C00673 V=800.0 PL=0
MOVL C00674 V=800.0 PL=0
MOVL C00675 V=800.0 PL=0
MOVL C00676 V=800.0 PL=0
MOVL C00677 V=800.0 PL=0
MOVL C00678 V=800.0 PL=0
MOVL C00679 V=800.0 PL=0
MOVL C00680 V=800.0 PL=0
MOVL C00681 V=800.0 PL=0
MOVL C00682 V=800.0 PL=0
MOVL C00683 V=800.0 PL=0
MOVL C00684 V=800.0 PL=0
MOVL C00685 V=800.0 PL=0
MOVL C00686 V=800.0 PL=0
MOVL C00687 V=800.0 PL=0
MOVL C00688 V=800.0 PL=0
MOVL C00689 V=800.0 PL=0
MOVL C00690 V=800.0 PL=0
MOVL C00691 V=800.0 PL=0
MOVL C00692 V=800.0 PL=0
MOVL C00693 V=800.0 PL=0
MOVL C00694 V=800.0 PL=0
MOVL C00695 V=800.0 PL=0
MOVL C00696 V=800.0 PL=0
MOVL C00697 V=800.0 PL=0
MOVL C00698 V=800.0 PL=0
MOVL C00699 V=800.0 PL=0
MOVL C00700 V=800.0 PL=0
MOVL C00701 V=800.0 PL=0
MOVL C00702 V=800.0 PL=0
MOVL C00703 V=800.0 PL=0
MOVL C00704 V=800.0 PL=0
MOVL C00705 V=800.0 PL=0
MOVL C00706 V=800.0 PL=0
MOVL C00707 V=800.0 PL=0
MOVL C00708 V=800.0 PL=0
MOVL C00709 V=800.0 PL=0
MOVL C00710 V=800.0 PL=0
MOVL C00711 V=800.0 PL=0
MOVL C00712 V=800.0 PL=0
MOVL C00713 V=800.0 PL=0
MOVL C00714 V=800.0 PL=0
MOVL C00715 V=800.0 PL=0
MOVL C00716 V=800.0 PL=0
MOVL C00717 V=800.0 PL=0
MOVL C00718 V=800.0 PL=0
MOVL C00719 V=800.0 PL=0
MOVL C00720 V=800.0 PL=0
MOVL C00721 V=800.0 PL=0
MOVL C00722 V=800.0 PL=0
MOVL C00723 V=800.0 PL=0
MOVL C00724 V=800.0 PL=0
MOVL C00725 V=800.0 PL=0
MOVL C00726 V=800.0 PL=0
MOVL C00727 V=800.0 PL=0
MOVL C00728 V=800.0 PL=0
MOVL C00729 V=800.0 PL=0
MOVL C00730 V=800.0 PL=0
MOVL C00731 V=800.0 PL=0
MOVL C00732 V=800.0 PL=0
MOVL C00733 V=800.0 PL=0
MOVL C00734 V=800.0 PL=0
MOVL C00735 V=800.0 PL=0
MOVL C00736 V=800.0 PL=0
MOVL C00737 V=800.0 PL=0
MOVL C00738 V=800.0 PL=0
MOVL C00739 V=800.0 PL=0
MOVL C00740 V=800.0 PL=0
MOVL C00741 V=800.0 PL=0
MOVL C00742 V=800.0 PL=0
MOVL C00743 V=800.0 PL=0
MOVL C00744 V=800.0 PL=0
MOVL C00745 V=800.0 PL=0
MOVL C00746 V=800.0 PL=0
MOVL C00747 V=800.0 PL=0
MOVL C00748 V=800.0 PL=0
MOVL C00749 V=800.0 PL=0
MOVL C00750 V=800.0 PL=0
MOVL C00751 V=800.0 PL=0
MOVL C00752 V=800.0 PL=0
MOVL C00753 V=800.0 PL=0
MOVL C00754 V=800.0 PL=0
MOVL C00755 V=800.0 PL=0
MOVL C00756 V=800.0 PL=0
MOVL C00757 V=800.0 PL=0
MOVL C00758 V=800.0 PL=0
MOVL C00759 V=800.0 PL=0
MOVL C00760 V=800.0 PL=0
MOVL C00761 V=800.0 PL=0
MOVL C00762 V=800.0 PL=0
MOVL C00763 V=800.0 PL=0
MOVL C00764 V=800.0 PL=0
MOVL C00765 V=800.0 PL=0
MOVL C00766 V=800.0 PL=0
MOVL C00767 V=800.0 PL=0
MOVL C00768 V=800.0 PL=0
MOVL C00769 V=800.0 PL=0
MOVL C00770 V=800.0 PL=0
MOVL C00771 V=800.0 PL=0
MOVL C00772 V=800.0 PL=0
MOVL C00773 V=800.0 PL=0
MOVL C00774 V=800.0 PL=0
MOVL C00775 V=800.0 PL=0
MOVL C00776 V=800.0 PL=0
MOVL C00777 V=800.0 PL=0
MOVL C00778 V=800.0 PL=0
MOVL C00779 V=800.0 PL=0
MOVL C00780 V=800.0 PL=0
MOVL C00781 V=800.0 PL=0
MOVL C00782 V=800.0 PL=0
MOVL C00783 V=800.0 PL=0
MOVL C00784 V=800.0 PL=0
MOVL C00785 V=800.0 PL=0
MOVL C00786 V=800.0 PL=0
MOVL C00787 V=800.0 PL=0
MOVL C00788 V=800.0 PL=0
MOVL C00789 V=800.0 PL=0
MOVL C00790 V=800.0 PL=0
MOVL C00791 V=800.0 PL=0
MOVL C00792 V=800.0 PL=0
MOVL C00793 V=800.0 PL=0
MOVL C00794 V=800.0 PL=0
MOVL C00795 V=800.0 PL=0
MOVL C00796 V=800.0 PL=0
MOVL C00797 V=800.0 PL=0
MOVL C00798 V=800.0 PL=0
MOVL C00799 V=800.0 PL=0
MOVL C00800 V=800.0 PL=0
MOVL C00801 V=800.0 PL=0
MOVL C00802 V=800.0 PL=0
MOVL C00803 V=800.0 PL=0
MOVL C00804 V=800.0 PL=0
MOVL C00805 V=800.0 PL=0
MOVL C00806 V=800.0 PL=0
MOVL C00807 V=800.0 PL=0
MOVL C00808 V=800.0 PL=0
MOVL C00809 V=800.0 PL=0
MOVL C00810 V=800.0 PL=0
MOVL C00811 V=800.0 PL=0
MOVL C00812 V=800.0 PL=0
MOVL C00813 V=800.0 PL=0
MOVL C00814 V=800.0 PL=0
MOVL C00815 V=800.0 PL=0
MOVL C00816 V=800.0 PL=0
MOVL C00817 V=800.0 PL=0
MOVL C00818 V=800.0 PL=0
MOVL C00819 V=800.0 PL=0
MOVL C00820 V=800.0 PL=0
MOVL C00821 V=800.0 PL=0
MOVL C00822 V=800.0 PL=0
MOVL C00823 V=800.0 PL=0
MOVL C00824 V=800.0 PL=0
MOVL C00825 V=800.0 PL=0
MOVL C00826 V=800.0 PL=0
MOVL C00827 V=800.0 PL=0
MOVL C00828 V=800.0 PL=0
MOVL C00829 V=800.0 PL=0
MOVL C00830 V=800.0 PL=0
MOVL C00831 V=800.0 PL=0
MOVL C00832 V=800.0 PL=0
MOVL C00833 V=800.0 PL=0
MOVL C00834 V=800.0 PL=0
MOVL C00835 V=800.0 PL=0
MOVL C00836 V=800.0 PL=0
MOVL C00837 V=800.0 PL=0
MOVL C00838 V=800.0 PL=0
MOVL C00839 V=800.0 PL=0
MOVL C00840 V=800.0 PL=0
MOVL C00841 V=800.0 PL=0
MOVL C00842 V=800.0 PL=0
MOVL C00843 V=800.0 PL=0
MOVL C00844 V=800.0 PL=0
MOVL C00845 V=800.0 PL=0
MOVL C00846 V=800.0 PL=0
MOVL C00847 V=800.0 PL=0
MOVL C00848 V=800.0 PL=0
MOVL C00849 V=800.0 PL=0
MOVL C00850 V=800.0 PL=0
MOVL C00851 V=800.0 PL=0
MOVL C00852 V=800.0 PL=0
MOVL C00853 V=800.0 PL=0
MOVL C00854 V=800.0 PL=0
MOVL C00855 V=800.0 PL=0
MOVL C00856 V=800.0 PL=0
MOVL C00857 V=800.0 PL=0
MOVL C00858 V=800.0 PL=0
MOVL C00859 V=800.0 PL=0
MOVL C00860 V=800.0 PL=0
MOVL C00861 V=800.0 PL=0
MOVL C00862 V=800.0 PL=0
MOVL C00863 V=800.0 PL=0
MOVL C00864 V=800.0 PL=0
MOVL C00865 V=800.0 PL=0
MOVL C00866 V=800.0 PL=0
MOVL C00867 V=800.0 PL=0
MOVL C00868 V=800.0 PL=0
MOVL C00869 V=800.0 PL=0
MOVL C00870 V=800.0 PL=0
MOVL C00871 V=800.0 PL=0
MOVL C00872 V=800.0 PL=0
MOVL C00873 V=800.0 PL=0
MOVL C00874 V=800.0 PL=0
MOVL C00875 V=800.0 PL=0
MOVL C00876 V=800.0 PL=0
MOVL C00877 V=800.0 PL=0
MOVL C00878 V=800.0 PL=0
MOVL C00879 V=800.0 PL=0
MOVL C00880 V=800.0 PL=0
MOVL C00881 V=800.0 PL=0
MOVL C00882 V=800.0 PL=0
MOVL C00883 V=800.0 PL=0
MOVL C00884 V=800.0 PL=0
MOVL C00885 V=800.0 PL=0
MOVL C00886 V=800.0 PL=0
MOVL C00887 V=800.0 PL=0
MOVL C00888 V=800.0 PL=0
MOVL C00889 V=800.0 PL=0
MOVL C00890 V=800.0 PL=0
MOVL C00891 V=800.0 PL=0
MOVL C00892 V=800.0 PL=0
MOVL C00893 V=800.0 PL=0
MOVL C00894 V=800.0 PL=0
MOVL C00895 V=800.0 PL=0
MOVL C00896 V=800.0 PL=0
MOVL C00897 V=800.0 PL=0
MOVL C00898 V=800.0 PL=0
MOVL C00899 V=800.0 PL=0
MOVL C00900 V=800.0 PL=0
MOVL C00901 V=800.0 PL=0
MOVL C00902 V=800.0 PL=0
MOVL C00903 V=800.0 PL=0
MOVL C00904 V=800.0 PL=0
MOVL C00905 V=800.0 PL=0
MOVL C00906 V=800.0 PL=0
MOVL C00907 V=800.0 PL=0
MOVL C00908 V=800.0 PL=0
MOVL C00909 V=800.0 PL=0
MOVL C00910 V=800.0 PL=0
MOVL C00911 V=800.0 PL=0
MOVL C00912 V=800.0 PL=0
MOVL C00913 V=800.0 PL=0
MOVL C00914 V=800.0 PL=0
MOVL C00915 V=800.0 PL=0
MOVL C00916 V=800.0 PL=0
MOVL C00917 V=800.0 PL=0
MOVL C00918 V=800.0 PL=0
MOVL C00919 V=800.0 PL=0
MOVL C00920 V=800.0 PL=0
MOVL C00921 V=800.0 PL=0
MOVL C00922 V=800.0 PL=0
MOVL C00923 V=800.0 PL=0
MOVL C00924 V=800.0 PL=0
MOVL C00925 V=800.0 PL=0
MOVL C00926 V=800.0 PL=0
MOVL C00927 V=800.0 PL=0
MOVL C00928 V=800.0 PL=0
MOVL C00929 V=800.0 PL=0
MOVL C00930 V=800.0 PL=0
MOVL C00931 V=800.0 PL=0
MOVL C00932 V=800.0 PL=0
MOVL C00933 V=800.0 PL=0
MOVL C00934 V=800.0 PL=0
MOVL C00935 V=800.0 PL=0
MOVL C00936 V=800.0 PL=0
MOVL C00937 V=800.0 PL=0
MOVL C00938 V=800.0 PL=0
MOVL C00939 V=800.0 PL=0
MOVL C00940 V=800.0 PL=0
MOVL C00941 V=800.0 PL=0
MOVL C00942 V=800.0 PL=0
MOVL C00943 V=800.0 PL=0
MOVL C00944 V=800.0 PL=0
MOVL C00945 V=800.0 PL=0
MOVL C00946 V=800.0 PL=0
MOVL C00947 V=800.0 PL=0
MOVL C00948 V=800.0 PL=0
MOVL C00949 V=800.0 PL=0
MOVL C00950 V=800.0 PL=0
MOVL C00951 V=800.0 PL=0
MOVL C00952 V=800.0 PL=0
MOVL C00953 V=800.0 PL=0
MOVL C00954 V=800.0 PL=0
MOVL C00955 V=800.0 PL=0
MOVL C00956 V=800.0 PL=0
MOVL C00957 V=800.0 PL=0
MOVL C00958 V=800.0 PL=0
MOVL C00959 V=800.0 PL=0
MOVL C00960 V=800.0 PL=0
MOVL C00961 V=800.0 PL=0
MOVL C00962 V=800.0 PL=0
MOVL C00963 V=800.0 PL=0
MOVL C00964 V=800.0 PL=0
MOVL C00965 V=800.0 PL=0
MOVL C00966 V=800.0 PL=0
MOVL C00967 V=800.0 PL=0
MOVL C00968 V=800.0 PL=0
MOVL C00969 V=800.0 PL=0
MOVL C00970 V=800.0 PL=0
MOVL C00971 V=800.0 PL=0
MOVL C00972 V=800.0 PL=0
MOVL C00973 V=800.0 PL=0
MOVL C00974 V=800.0 PL=0
MOVL C00975 V=800.0 PL=0
MOVL C00976 V=800.0 PL=0
MOVL C00977 V=800.0 PL=0
MOVL C00978 V=800.0 PL=0
MOVL C00979 V=800.0 PL=0
MOVL C00980 V=800.0 PL=0
MOVL C00981 V=800.0 PL=0
MOVL C00982 V=800.0 PL=0
MOVL C00983 V=800.0 PL=0
MOVL C00984 V=800.0 PL=0
MOVL C00985 V=800.0 PL=0
MOVL C00986 V=800.0 PL=0
MOVL C00987 V=800.0 PL=0
MOVL C00988 V=800.0 PL=0
MOVL C00989 V=800.0 PL=0
MOVL C00990 V=800.0 PL=0
MOVL C00991 V=800.0 PL=0
MOVL C00992 V=800.0 PL=0
MOVL C00993 V=800.0 PL=0
MOVL C00994 V=800.0 PL=0
MOVL C00995 V=800.0 PL=0
MOVL C00996 V=800.0 PL=0
MOVL C00997 V=800.0 PL=0
MOVL C00998 V=800.0 PL=0
MOVL C00999 V=800.0 PL=0
MOVL C01000 V=800.0 PL=0
MOVL C01001 V=800.0 PL=0
MOVL C01002 V=800.0 PL=0
MOVL C01003 V=800.0 PL=0
MOVL C01004 V=800.0 PL=0
MOVL C01005 V=800.0 PL=0
MOVL C01006 V=800.0 PL=0
MOVL C01007 V=800.0 PL=0
MOVL C01008 V=800.0 PL=0
MOVL C01009 V=800.0 PL=0
MOVL C01010 V=800.0 PL=0
MOVL C01011 V=800.0 PL=0
MOVL C01012 V=800.0 PL=0
MOVL C01013 V=800.0 PL=0
MOVL C01014 V=800.0 PL=0
MOVL C01015 V=800.0 PL=0
MOVL C01016 V=800.0 PL=0
MOVL C01017 V=800.0 PL=0
MOVL C01018 V=800.0 PL=0
MOVL C01019 V=800.0 PL=0
MOVL C01020 V=800.0 PL=0
MOVL C01021 V=800.0 PL=0
MOVL C01022 V=800.0 PL=0
MOVL C01023 V=800.0 PL=0
MOVL C01024 V=800.0 PL=0
MOVL C01025 V=800.0 PL=0
MOVL C01026 V=800.0 PL=0
MOVL C01027 V=800.0 PL=0
MOVL C01028 V=800.0 PL=0
MOVL C01029 V=800.0 PL=0
MOVL C01030 V=800.0 PL=0
MOVL C01031 V=800.0 PL=0
MOVL C01032 V=800.0 PL=0
MOVL C01033 V=800.0 PL=0
MOVL C01034 V=800.0 PL=0
MOVL C01035 V=800.0 PL=0
MOVL C01036 V=800.0 PL=0
MOVL C01037 V=800.0 PL=0
MOVL C01038 V=800.0 PL=0
MOVL C01039 V=800.0 PL=0
MOVL C01040 V=800.0 PL=0
MOVL C01041 V=800.0 PL=0
MOVL C01042 V=800.0 PL=0
MOVL C01043 V=800.0 PL=0
MOVL C01044 V=800.0 PL=0
MOVL C01045 V=800.0 PL=0
MOVL C01046 V=800.0 PL=0
MOVL C01047 V=800.0 PL=0
MOVL C01048 V=800.0 PL=0
MOVL C01049 V=800.0 PL=0
MOVL C01050 V=800.0 PL=0
MOVL C01051 V=800.0 PL=0
MOVL C01052 V=800.0 PL=0
MOVL C01053 V=800.0 PL=0
MOVL C01054 V=800.0 PL=0
MOVL C01055 V=800.0 PL=0
MOVL C01056 V=800.0 PL=0
MOVL C01057 V=800.0 PL=0
MOVL C01058 V=800.0 PL=0
MOVL C01059 V=800.0 PL=0
MOVL C01060 V=800.0 PL=0
MOVL C01061 V=800.0 PL=0
MOVL C01062 V=800.0 PL=0
MOVL C01063 V=800.0 PL=0
MOVL C01064 V=800.0 PL=0
MOVL C01065 V=800.0 PL=0
MOVL C01066 V=800.0 PL=0
MOVL C01067 V=800.0 PL=0
MOVL C01068 V=800.0 PL=0
MOVL C01069 V=800.0 PL=0
MOVL C01070 V=800.0 PL=0
MOVL C01071 V=800.0 PL=0
MOVL C01072 V=800.0 PL=0
MOVL C01073 V=800.0 PL=0
MOVL C01074 V=800.0 PL=0
MOVL C01075 V=800.0 PL=0
MOVL C01076 V=800.0 PL=0
MOVL C01077 V=800.0 PL=0
MOVL C01078 V=800.0 PL=0
MOVL C01079 V=800.0 PL=0
MOVL C01080 V=800.0 PL=0
MOVL C01081 V=800.0 PL=0
MOVL C01082 V=800.0 PL=0
MOVL C01083 V=800.0 PL=0
MOVL C01084 V=800.0 PL=0
MOVL C01085 V=800.0 PL=0
MOVL C01086 V=800.0 PL=0
MOVL C01087 V=800.0 PL=0
MOVL C01088 V=800.0 PL=0
MOVL C01089 V=800.0 PL=0
MOVL C01090 V=800.0 PL=0
MOVL C01091 V=800.0 PL=0
MOVL C01092 V=800.0 PL=0
MOVL C01093 V=800.0 PL=0
MOVL C01094 V=800.0 PL=0
MOVL C01095 V=800.0 PL=0
MOVL C01096 V=800.0 PL=0
MOVL C01097 V=800.0 PL=0
MOVL C01098 V=800.0 PL=0
MOVL C01099 V=800.0 PL=0
MOVL C01100 V=800.0 PL=0
MOVL C01101 V=800.0 PL=0
MOVL C01102 V=800.0 PL=0
MOVL C01103 V=800.0 PL=0
MOVL C01104 V=800.0 PL=0
MOVL C01105 V=800.0 PL=0
MOVL C01106 V=800.0 PL=0
MOVL C01107 V=800.0 PL=0
MOVL C01108 V=800.0 PL=0
MOVL C01109 V=800.0 PL=0
MOVL C01110 V=800.0 PL=0
MOVL C01111 V=800.0 PL=0
MOVL C01112 V=800.0 PL=0
MOVL C01113 V=800.0 PL=0
MOVL C01114 V=800.0 PL=0
MOVL C01115 V=800.0 PL=0
MOVL C01116 V=800.0 PL=0
MOVL C01117 V=800.0 PL=0
MOVL C01118 V=800.0 PL=0
MOVL C01119 V=800.0 PL=0
MOVL C01120 V=800.0 PL=0
MOVL C01121 V=800.0 PL=0
MOVL C01122 V=800.0 PL=0
MOVL C01123 V=800.0 PL=0
MOVL C01124 V=800.0 PL=0
MOVL C01125 V=800.0 PL=0
MOVL C01126 V=800.0 PL=0
MOVL C01127 V=800.0 PL=0
MOVL C01128 V=800.0 PL=0
MOVL C01129 V=800.0 PL=0
MOVL C01130 V=800.0 PL=0
MOVL C01131 V=800.0 PL=0
MOVL C01132 V=800.0 PL=0
MOVL C01133 V=800.0 PL=0
MOVL C01134 V=800.0 PL=0
MOVL C01135 V=800.0 PL=0
MOVL C01136 V=800.0 PL=0
MOVL C01137 V=800.0 PL=0
MOVL C01138 V=800.0 PL=0
MOVL C01139 V=800.0 PL=0
MOVL C01140 V=800.0 PL=0
MOVL C01141 V=800.0 PL=0
MOVL C01142 V=800.0 PL=0
MOVL C01143 V=800.0 PL=0
MOVL C01144 V=800.0 PL=0
MOVL C01145 V=800.0 PL=0
MOVL C01146 V=800.0 PL=0
MOVL C01147 V=800.0 PL=0
MOVL C01148 V=800.0 PL=0
MOVL C01149 V=800.0 PL=0
MOVL C01150 V=800.0 PL=0
MOVL C01151 V=800.0 PL=0
MOVL C01152 V=800.0 PL=0
MOVL C01153 V=800.0 PL=0
MOVL C01154 V=800.0 PL=0
MOVL C01155 V=800.0 PL=0
MOVL C01156 V=800.0 PL=0
MOVL C01157 V=800.0 PL=0
MOVL C01158 V=800.0 PL=0
MOVL C01159 V=800.0 PL=0
MOVL C01160 V=800.0 PL=0
MOVL C01161 V=800.0 PL=0
MOVL C01162 V=800.0 PL=0
MOVL C01163 V=800.0 PL=0
MOVL C01164 V=800.0 PL=0
MOVL C01165 V=800.0 PL=0
MOVL C01166 V=800.0 PL=0
MOVL C01167 V=800.0 PL=0
MOVL C01168 V=800.0 PL=0
MOVL C01169 V=800.0 PL=0
MOVL C01170 V=800.0 PL=0
MOVL C01171 V=800.0 PL=0
MOVL C01172 V=800.0 PL=0
MOVL C01173 V=800.0 PL=0
MOVL C01174 V=800.0 PL=0
MOVL C01175 V=800.0 PL=0
MOVL C01176 V=800.0 PL=0
MOVL C01177 V=800.0 PL=0
MOVL C01178 V=800.0 PL=0
MOVL C01179 V=800.0 PL=0
MOVL C01180 V=800.0 PL=0
MOVL C01181 V=800.0 PL=0
MOVL C01182 V=800.0 PL=0
MOVL C01183 V=800.0 PL=0
MOVL C01184 V=800.0 PL=0
MOVL C01185 V=800.0 PL=0
MOVL C01186 V=800.0 PL=0
MOVL C01187 V=800.0 PL=0
MOVL C01188 V=800.0 PL=0
MOVL C01189 V=800.0 PL=0
MOVL C01190 V=800.0 PL=0
MOVL C01191 V=800.0 PL=0
MOVL C01192 V=800.0 PL=0
MOVL C01193 V=800.0 PL=0
MOVL C01194 V=800.0 PL=0
MOVL C01195 V=800.0 PL=0
MOVL C01196 V=800.0 PL=0
MOVL C01197 V=800.0 PL=0
MOVL C01198 V=800.0 PL=0
MOVL C01199 V=800.0 PL=0
MOVL C01200 V=800.0 PL=0
MOVL C01201 V=800.0 PL=0
MOVL C01202 V=800.0 PL=0
MOVL C01203 V=800.0 PL=0
MOVL C01204 V=800.0 PL=0
MOVL C01205 V=800.0 PL=0
MOVL C01206 V=800.0 PL=0
MOVL C01207 V=800.0 PL=0
MOVL C01208 V=800.0 PL=0
MOVL C01209 V=800.0 PL=0
MOVL C01210 V=800.0 PL=0
MOVL C01211 V=800.0 PL=0
MOVL C01212 V=800.0 PL=0
MOVL C01213 V=800.0 PL=0
MOVL C01214 V=800.0 PL=0
MOVL C01215 V=800.0 PL=0
MOVL C01216 V=800.0 PL=0
MOVL C01217 V=800.0 PL=0
MOVL C01218 V=800.0 PL=0
MOVL C01219 V=800.0 PL=0
MOVL C01220 V=800.0 PL=0
MOVL C01221 V=800.0 PL=0
MOVL C01222 V=800.0 PL=0
MOVL C01223 V=800.0 PL=0
MOVL C01224 V=800.0 PL=0
MOVL C01225 V=800.0 PL=0
MOVL C01226 V=800.0 PL=0
MOVL C01227 V=800.0 PL=0
MOVL C01228 V=800.0 PL=0
MOVL C01229 V=800.0 PL=0
MOVL C01230 V=800.0 PL=0
MOVL C01231 V=800.0 PL=0
MOVL C01232 V=800.0 PL=0
MOVL C01233 V=800.0 PL=0
MOVL C01234 V=800.0 PL=0
MOVL C01235 V=800.0 PL=0
MOVL C01236 V=800.0 PL=0
MOVL C01237 V=800.0 PL=0
MOVL C01238 V=800.0 PL=0
MOVL C01239 V=800.0 PL=0
MOVL C01240 V=800.0 PL=0
MOVL C01241 V=800.0 PL=0
MOVL C01242 V=800.0 PL=0
MOVL C01243 V=800.0 PL=0
MOVL C01244 V=800.0 PL=0
MOVL C01245 V=800.0 PL=0
MOVL C01246 V=800.0 PL=0
MOVL C01247 V=800.0 PL=0
MOVL C01248 V=800.0 PL=0
MOVL C01249 V=800.0 PL=0
MOVL C01250 V=800.0 PL=0
MOVL C01251 V=800.0 PL=0
MOVL C01252 V=800.0 PL=0
MOVL C01253 V=800.0 PL=0
MOVL C01254 V=800.0 PL=0
MOVL C01255 V=800.0 PL=0
MOVL C01256 V=800.0 PL=0
MOVL C01257 V=800.0 PL=0
MOVL C01258 V=800.0 PL=0
MOVL C01259 V=800.0 PL=0
MOVL C01260 V=800.0 PL=0
MOVL C01261 V=800.0 PL=0
MOVL C01262 V=800.0 PL=0
MOVL C01263 V=800.0 PL=0
MOVL C01264 V=800.0 PL=0
MOVL C01265 V=800.0 PL=0
MOVL C01266 V=800.0 PL=0
MOVL C01267 V=800.0 PL=0
MOVL C01268 V=800.0 PL=0
MOVL C01269 V=800.0 PL=0
MOVL C01270 V=800.0 PL=0
MOVL C01271 V=800.0 PL=0
MOVL C01272 V=800.0 PL=0
MOVL C01273 V=800.0 PL=0
MOVL C01274 V=800.0 PL=0
MOVL C01275 V=800.0 PL=0
MOVL C01276 V=800.0 PL=0
MOVL C01277 V=800.0 PL=0
MOVL C01278 V=800.0 PL=0
MOVL C01279 V=800.0 PL=0
MOVL C01280 V=800.0 PL=0
MOVL C01281 V=800.0 PL=0
MOVL C01282 V=800.0 PL=0
MOVL C01283 V=800.0 PL=0
MOVL C01284 V=800.0 PL=0
MOVL C01285 V=800.0 PL=0
MOVL C01286 V=800.0 PL=0
MOVL C01287 V=800.0 PL=0
MOVL C01288 V=800.0 PL=0
MOVL C01289 V=800.0 PL=0
MOVL C01290 V=800.0 PL=0
MOVL C01291 V=800.0 PL=0
MOVL C01292 V=800.0 PL=0
MOVL C01293 V=800.0 PL=0
MOVL C01294 V=800.0 PL=0
MOVL C01295 V=800.0 PL=0
MOVL C01296 V=800.0 PL=0
MOVL C01297 V=800.0 PL=0
MOVL C01298 V=800.0 PL=0
MOVL C01299 V=800.0 PL=0
MOVL C01300 V=800.0 PL=0
MOVL C01301 V=800.0 PL=0
MOVL C01302 V=800.0 PL=0
MOVL C01303 V=800.0 PL=0
MOVL C01304 V=800.0 PL=0
MOVL C01305 V=800.0 PL=0
MOVL C01306 V=800.0 PL=0
MOVL C01307 V=800.0 PL=0
MOVL C01308 V=800.0 PL=0
MOVL C01309 V=800.0 PL=0
MOVL C01310 V=800.0 PL=0
MOVL C01311 V=800.0 PL=0
MOVL C01312 V=800.0 PL=0
MOVL C01313 V=800.0 PL=0
MOVL C01314 V=800.0 PL=0
MOVL C01315 V=800.0 PL=0
MOVL C01316 V=800.0 PL=0
MOVL C01317 V=800.0 PL=0
MOVL C01318 V=800.0 PL=0
MOVL C01319 V=800.0 PL=0
MOVL C01320 V=800.0 PL=0
MOVL C01321 V=800.0 PL=0
MOVL C01322 V=800.0 PL=0
MOVL C01323 V=800.0 PL=0
MOVL C01324 V=800.0 PL=0
MOVL C01325 V=800.0 PL=0
MOVL C01326 V=800.0 PL=0
MOVL C01327 V=800.0 PL=0
MOVL C01328 V=800.0 PL=0
MOVL C01329 V=800.0 PL=0
MOVL C01330 V=800.0 PL=0
MOVL C01331 V=800.0 PL=0
MOVL C01332 V=800.0 PL=0
MOVL C01333 V=800.0 PL=0
MOVL C01334 V=800.0 PL=0
MOVL C01335 V=800.0 PL=0
MOVL C01336 V=800.0 PL=0
MOVL C01337 V=800.0 PL=0
MOVL C01338 V=800.0 PL=0
MOVL C01339 V=800.0 PL=0
MOVL C01340 V=800.0 PL=0
MOVL C01341 V=800.0 PL=0
MOVL C01342 V=800.0 PL=0
MOVL C01343 V=800.0 PL=0
MOVL C01344 V=800.0 PL=0
MOVL C01345 V=800.0 PL=0
MOVL C01346 V=800.0 PL=0
MOVL C01347 V=800.0 PL=0
MOVL C01348 V=800.0 PL=0
MOVL C01349 V=800.0 PL=0
MOVL C01350 V=800.0 PL=0
MOVL C01351 V=800.0 PL=0
MOVL C01352 V=800.0 PL=0
MOVL C01353 V=800.0 PL=0
MOVL C01354 V=800.0 PL=0
MOVL C01355 V=800.0 PL=0
MOVL C01356 V=800.0 PL=0
MOVL C01357 V=800.0 PL=0
MOVL C01358 V=800.0 PL=0
MOVL C01359 V=800.0 PL=0
MOVL C01360 V=800.0 PL=0
MOVL C01361 V=800.0 PL=0
MOVL C01362 V=800.0 PL=0
MOVL C01363 V=800.0 PL=0
MOVL C01364 V=800.0 PL=0
MOVL C01365 V=800.0 PL=0
MOVL C01366 V=800.0 PL=0
MOVL C01367 V=800.0 PL=0
MOVL C01368 V=800.0 PL=0
MOVL C01369 V=800.0 PL=0
MOVL C01370 V=800.0 PL=0
MOVL C01371 V=800.0 PL=0
MOVL C01372 V=800.0 PL=0
MOVL C01373 V=800.0 PL=0
MOVL C01374 V=800.0 PL=0
MOVL C01375 V=800.0 PL=0
MOVL C01376 V=800.0 PL=0
MOVL C01377 V=800.0 PL=0
MOVL C01378 V=800.0 PL=0
MOVL C01379 V=800.0 PL=0
MOVL C01380 V=800.0 PL=0
MOVL C01381 V=800.0 PL=0
MOVL C01382 V=800.0 PL=0
MOVL C01383 V=800.0 PL=0
MOVL C01384 V=800.0 PL=0
MOVL C01385 V=800.0 PL=0
MOVL C01386 V=800.0 PL=0
MOVL C01387 V=800.0 PL=0
MOVL C01388 V=800.0 PL=0
MOVL C01389 V=800.0 PL=0
MOVL C01390 V=800.0 PL=0
MOVL C01391 V=800.0 PL=0
MOVL C01392 V=800.0 PL=0
MOVL C01393 V=800.0 PL=0
MOVL C01394 V=800.0 PL=0
MOVL C01395 V=800.0 PL=0
MOVL C01396 V=800.0 PL=0
MOVL C01397 V=800.0 PL=0
MOVL C01398 V=800.0 PL=0
MOVL C01399 V=800.0 PL=0
MOVL C01400 V=800.0 PL=0
MOVL C01401 V=800.0 PL=0
MOVL C01402 V=800.0 PL=0
MOVL C01403 V=800.0 PL=0
MOVL C01404 V=800.0 PL=0
MOVL C01405 V=800.0 PL=0
MOVL C01406 V=800.0 PL=0
MOVL C01407 V=800.0 PL=0
MOVL C01408 V=800.0 PL=0
MOVL C01409 V=800.0 PL=0
MOVL C01410 V=800.0 PL=0
MOVL C01411 V=800.0 PL=0
MOVL C01412 V=800.0 PL=0
MOVL C01413 V=800.0 PL=0
MOVL C01414 V=800.0 PL=0
MOVL C01415 V=800.0 PL=0
MOVL C01416 V=800.0 PL=0
MOVL C01417 V=800.0 PL=0
MOVL C01418 V=800.0 PL=0
MOVL C01419 V=800.0 PL=0
MOVL C01420 V=800.0 PL=0
MOVL C01421 V=800.0 PL=0
MOVL C01422 V=800.0 PL=0
MOVL C01423 V=800.0 PL=0
MOVL C01424 V=800.0 PL=0
MOVL C01425 V=800.0 PL=0
MOVL C01426 V=800.0 PL=0
MOVL C01427 V=800.0 PL=0
MOVL C01428 V=800.0 PL=0
MOVL C01429 V=800.0 PL=0
MOVL C01430 V=800.0 PL=0
MOVL C01431 V=800.0 PL=0
MOVL C01432 V=800.0 PL=0
MOVL C01433 V=800.0 PL=0
MOVL C01434 V=800.0 PL=0
MOVL C01435 V=800.0 PL=0
MOVL C01436 V=800.0 PL=0
MOVL C01437 V=800.0 PL=0
MOVL C01438 V=800.0 PL=0
MOVL C01439 V=800.0 PL=0
MOVL C01440 V=800.0 PL=0
MOVL C01441 V=800.0 PL=0
MOVL C01442 V=800.0 PL=0
MOVL C01443 V=800.0 PL=0
MOVL C01444 V=800.0 PL=0
MOVL C01445 V=800.0 PL=0
MOVL C01446 V=800.0 PL=0
MOVL C01447 V=800.0 PL=0
MOVL C01448 V=800.0 PL=0
MOVL C01449 V=800.0 PL=0
MOVL C01450 V=800.0 PL=0
MOVL C01451 V=800.0 PL=0
MOVL C01452 V=800.0 PL=0
MOVL C01453 V=800.0 PL=0
MOVL C01454 V=800.0 PL=0
MOVL C01455 V=800.0 PL=0
MOVL C01456 V=800.0 PL=0
MOVL C01457 V=800.0 PL=0
MOVL C01458 V=800.0 PL=0
MOVL C01459 V=800.0 PL=0
MOVL C01460 V=800.0 PL=0
MOVL C01461 V=800.0 PL=0
MOVL C01462 V=800.0 PL=0
MOVL C01463 V=800.0 PL=0
MOVL C01464 V=800.0 PL=0
MOVL C01465 V=800.0 PL=0
MOVL C01466 V=800.0 PL=0
MOVL C01467 V=800.0 PL=0
MOVL C01468 V=800.0 PL=0
MOVL C01469 V=800.0 PL=0
MOVL C01470 V=800.0 PL=0
MOVL C01471 V=800.0 PL=0
MOVL C01472 V=800.0 PL=0
MOVL C01473 V=800.0 PL=0
MOVL C01474 V=800.0 PL=0
MOVL C01475 V=800.0 PL=0
MOVL C01476 V=800.0 PL=0
MOVL C01477 V=800.0 PL=0
MOVL C01478 V=800.0 PL=0
MOVL C01479 V=800.0 PL=0
MOVL C01480 V=800.0 PL=0
MOVL C01481 V=800.0 PL=0
MOVL C01482 V=800.0 PL=0
MOVL C01483 V=800.0 PL=0
MOVL C01484 V=800.0 PL=0
MOVL C01485 V=800.0 PL=0
MOVL C01486 V=800.0 PL=0
MOVL C01487 V=800.0 PL=0
MOVL C01488 V=800.0 PL=0
MOVL C01489 V=800.0 PL=0
MOVL C01490 V=800.0 PL=0
MOVL C01491 V=800.0 PL=0
MOVL C01492 V=800.0 PL=0
MOVL C01493 V=800.0 PL=0
MOVL C01494 V=800.0 PL=0
MOVL C01495 V=800.0 PL=0
MOVL C01496 V=800.0 PL=0
MOVL C01497 V=800.0 PL=0
MOVL C01498 V=800.0 PL=0
MOVL C01499 V=800.0 PL=0
MOVL C01500 V=800.0 PL=0
MOVL C01501 V=800.0 PL=0
MOVL C01502 V=800.0 PL=0
MOVL C01503 V=800.0 PL=0
MOVL C01504 V=800.0 PL=0
MOVL C01505 V=800.0 PL=0
MOVL C01506 V=800.0 PL=0
MOVL C01507 V=800.0 PL=0
MOVL C01508 V=800.0 PL=0
MOVL C01509 V=800.0 PL=0
MOVL C01510 V=800.0 PL=0
MOVL C01511 V=800.0 PL=0
MOVL C01512 V=800.0 PL=0
MOVL C01513 V=800.0 PL=0
MOVL C01514 V=800.0 PL=0
MOVL C01515 V=800.0 PL=0
MOVL C01516 V=800.0 PL=0
MOVL C01517 V=800.0 PL=0
MOVL C01518 V=800.0 PL=0
MOVL C01519 V=800.0 PL=0
MOVL C01520 V=800.0 PL=0
MOVL C01521 V=800.0 PL=0
MOVL C01522 V=800.0 PL=0
MOVL C01523 V=800.0 PL=0
MOVL C01524 V=800.0 PL=0
MOVL C01525 V=800.0 PL=0
MOVL C01526 V=800.0 PL=0
MOVL C01527 V=800.0 PL=0
MOVL C01528 V=800.0 PL=0
MOVL C01529 V=800.0 PL=0
MOVL C01530 V=800.0 PL=0
MOVL C01531 V=800.0 PL=0
MOVL C01532 V=800.0 PL=0
MOVL C01533 V=800.0 PL=0
MOVL C01534 V=800.0 PL=0
MOVL C01535 V=800.0 PL=0
MOVL C01536 V=800.0 PL=0
MOVL C01537 V=800.0 PL=0
MOVL C01538 V=800.0 PL=0
MOVL C01539 V=800.0 PL=0
MOVL C01540 V=800.0 PL=0
MOVL C01541 V=800.0 PL=0
MOVL C01542 V=800.0 PL=0
MOVL C01543 V=800.0 PL=0
MOVL C01544 V=800.0 PL=0
MOVL C01545 V=800.0 PL=0
MOVL C01546 V=800.0 PL=0
MOVL C01547 V=800.0 PL=0
MOVL C01548 V=800.0 PL=0
MOVL C01549 V=800.0 PL=0
MOVL C01550 V=800.0 PL=0
MOVL C01551 V=800.0 PL=0
MOVL C01552 V=800.0 PL=0
MOVL C01553 V=800.0 PL=0
MOVL C01554 V=800.0 PL=0
MOVL C01555 V=800.0 PL=0
MOVL C01556 V=800.0 PL=0
MOVL C01557 V=800.0 PL=0
MOVL C01558 V=800.0 PL=0
MOVL C01559 V=800.0 PL=0
MOVL C01560 V=800.0 PL=0
MOVL C01561 V=800.0 PL=0
MOVL C01562 V=800.0 PL=0
MOVL C01563 V=800.0 PL=0
MOVL C01564 V=800.0 PL=0
MOVL C01565 V=800.0 PL=0
MOVL C01566 V=800.0 PL=0
MOVL C01567 V=800.0 PL=0
MOVL C01568 V=800.0 PL=0
MOVL C01569 V=800.0 PL=0
MOVL C01570 V=800.0 PL=0
MOVL C01571 V=800.0 PL=0
MOVL C01572 V=800.0 PL=0
MOVL C01573 V=800.0 PL=0
MOVL C01574 V=800.0 PL=0
MOVL C01575 V=800.0 PL=0
MOVL C01576 V=800.0 PL=0
MOVL C01577 V=800.0 PL=0
MOVL C01578 V=800.0 PL=0
MOVL C01579 V=800.0 PL=0
MOVL C01580 V=800.0 PL=0
MOVL C01581 V=800.0 PL=0
MOVL C01582 V=800.0 PL=0
MOVL C01583 V=800.0 PL=0
MOVL C01584 V=800.0 PL=0
MOVL C01585 V=800.0 PL=0
MOVL C01586 V=800.0 PL=0
MOVL C01587 V=800.0 PL=0
MOVL C01588 V=800.0 PL=0
MOVL C01589 V=800.0 PL=0
MOVL C01590 V=800.0 PL=0
MOVL C01591 V=800.0 PL=0
MOVL C01592 V=800.0 PL=0
MOVL C01593 V=800.0 PL=0
MOVL C01594 V=800.0 PL=0
MOVL C01595 V=800.0 PL=0
MOVL C01596 V=800.0 PL=0
MOVL C01597 V=800.0 PL=0
MOVL C01598 V=800.0 PL=0
MOVL C01599 V=800.0 PL=0
MOVL C01600 V=800.0 PL=0
MOVL C01601 V=800.0 PL=0
MOVL C01602 V=800.0 PL=0
MOVL C01603 V=800.0 PL=0
MOVL C01604 V=800.0 PL=0
MOVL C01605 V=800.0 PL=0
MOVL C01606 V=800.0 PL=0
MOVL C01607 V=800.0 PL=0
MOVL C01608 V=800.0 PL=0
MOVL C01609 V=800.0 PL=0
MOVL C01610 V=800.0 PL=0
MOVL C01611 V=800.0 PL=0
MOVL C01612 V=800.0 PL=0
MOVL C01613 V=800.0 PL=0
MOVL C01614 V=800.0 PL=0
MOVL C01615 V=800.0 PL=0
MOVL C01616 V=800.0 PL=0
MOVL C01617 V=800.0 PL=0
MOVL C01618 V=800.0 PL=0
MOVL C01619 V=800.0 PL=0
MOVL C01620 V=800.0 PL=0
MOVL C01621 V=800.0 PL=0
MOVL C01622 V=800.0 PL=0
MOVL C01623 V=800.0 PL=0
MOVL C01624 V=800.0 PL=0
MOVL C01625 V=800.0 PL=0
MOVL C01626 V=800.0 PL=0
MOVL C01627 V=800.0 PL=0
MOVL C01628 V=800.0 PL=0
MOVL C01629 V=800.0 PL=0
MOVL C01630 V=800.0 PL=0
MOVL C01631 V=800.0 PL=0
MOVL C01632 V=800.0 PL=0
MOVL C01633 V=800.0 PL=0
MOVL C01634 V=800.0 PL=0
MOVL C01635 V=800.0 PL=0
MOVL C01636 V=800.0 PL=0
MOVL C01637 V=800.0 PL=0
MOVL C01638 V=800.0 PL=0
MOVL C01639 V=800.0 PL=0
MOVL C01640 V=800.0 PL=0
MOVL C01641 V=800.0 PL=0
MOVL C01642 V=800.0 PL=0
MOVL C01643 V=800.0 PL=0
MOVL C01644 V=800.0 PL=0
MOVL C01645 V=800.0 PL=0
MOVL C01646 V=800.0 PL=0
MOVL C01647 V=800.0 PL=0
MOVL C01648 V=800.0 PL=0
MOVL C01649 V=800.0 PL=0
MOVL C01650 V=800.0 PL=0
MOVL C01651 V=800.0 PL=0
MOVL C01652 V=800.0 PL=0
MOVL C01653 V=800.0 PL=0
MOVL C01654 V=800.0 PL=0
MOVL C01655 V=800.0 PL=0
MOVL C01656 V=800.0 PL=0
MOVL C01657 V=800.0 PL=0
MOVL C01658 V=800.0 PL=0
MOVL C01659 V=800.0 PL=0
MOVL C01660 V=800.0 PL=0
MOVL C01661 V=800.0 PL=0
MOVL C01662 V=800.0 PL=0
MOVL C01663 V=800.0 PL=0
MOVL C01664 V=800.0 PL=0
MOVL C01665 V=800.0 PL=0
MOVL C01666 V=800.0 PL=0
MOVL C01667 V=800.0 PL=0
MOVL C01668 V=800.0 PL=0
MOVL C01669 V=800.0 PL=0
MOVL C01670 V=800.0 PL=0
MOVL C01671 V=800.0 PL=0
MOVL C01672 V=800.0 PL=0
MOVL C01673 V=800.0 PL=0
MOVL C01674 V=800.0 PL=0
MOVL C01675 V=800.0 PL=0
MOVL C01676 V=800.0 PL=0
MOVL C01677 V=800.0 PL=0
MOVL C01678 V=800.0 PL=0
MOVL C01679 V=800.0 PL=0
MOVL C01680 V=800.0 PL=0
MOVL C01681 V=800.0 PL=0
MOVL C01682 V=800.0 PL=0
MOVL C01683 V=800.0 PL=0
MOVL C01684 V=800.0 PL=0
MOVL C01685 V=800.0 PL=0
MOVL C01686 V=800.0 PL=0
MOVL C01687 V=800.0 PL=0
MOVL C01688 V=800.0 PL=0
MOVL C01689 V=800.0 PL=0
MOVL C01690 V=800.0 PL=0
MOVL C01691 V=800.0 PL=0
MOVL C01692 V=800.0 PL=0
MOVL C01693 V=800.0 PL=0
MOVL C01694 V=800.0 PL=0
MOVL C01695 V=800.0 PL=0
MOVL C01696 V=800.0 PL=0
MOVL C01697 V=800.0 PL=0
MOVL C01698 V=800.0 PL=0
MOVL C01699 V=800.0 PL=0
MOVL C01700 V=800.0 PL=0
MOVL C01701 V=800.0 PL=0
MOVL C01702 V=800.0 PL=0
MOVL C01703 V=800.0 PL=0
MOVL C01704 V=800.0 PL=0
MOVL C01705 V=800.0 PL=0
MOVL C01706 V=800.0 PL=0
MOVL C01707 V=800.0 PL=0
MOVL C01708 V=800.0 PL=0
MOVL C01709 V=800.0 PL=0
MOVL C01710 V=800.0 PL=0
MOVL C01711 V=800.0 PL=0
MOVL C01712 V=800.0 PL=0
MOVL C01713 V=800.0 PL=0
MOVL C01714 V=800.0 PL=0
MOVL C01715 V=800.0 PL=0
MOVL C01716 V=800.0 PL=0
MOVL C01717 V=800.0 PL=0
MOVL C01718 V=800.0 PL=0
MOVL C01719 V=800.0 PL=0
MOVL C01720 V=800.0 PL=0
MOVL C01721 V=800.0 PL=0
MOVL C01722 V=800.0 PL=0
MOVL C01723 V=800.0 PL=0
MOVL C01724 V=800.0 PL=0
MOVL C01725 V=800.0 PL=0
MOVL C01726 V=800.0 PL=0
MOVL C01727 V=800.0 PL=0
MOVL C01728 V=800.0 PL=0
MOVL C01729 V=800.0 PL=0
MOVL C01730 V=800.0 PL=0
MOVL C01731 V=800.0 PL=0
MOVL C01732 V=800.0 PL=0
MOVL C01733 V=800.0 PL=0
MOVL C01734 V=800.0 PL=0
MOVL C01735 V=800.0 PL=0
MOVL C01736 V=800.0 PL=0
MOVL C01737 V=800.0 PL=0
MOVL C01738 V=800.0 PL=0
MOVL C01739 V=800.0 PL=0
MOVL C01740 V=800.0 PL=0
MOVL C01741 V=800.0 PL=0
MOVL C01742 V=800.0 PL=0
MOVL C01743 V=800.0 PL=0
MOVL C01744 V=800.0 PL=0
MOVL C01745 V=800.0 PL=0
MOVL C01746 V=800.0 PL=0
MOVL C01747 V=800.0 PL=0
MOVL C01748 V=800.0 PL=0
MOVL C01749 V=800.0 PL=0
MOVL C01750 V=800.0 PL=0
MOVL C01751 V=800.0 PL=0
MOVL C01752 V=800.0 PL=0
MOVL C01753 V=800.0 PL=0
MOVL C01754 V=800.0 PL=0
MOVL C01755 V=800.0 PL=0
MOVL C01756 V=800.0 PL=0
MOVL C01757 V=800.0 PL=0
MOVL C01758 V=800.0 PL=0
MOVL C01759 V=800.0 PL=0
MOVL C01760 V=800.0 PL=0
MOVL C01761 V=800.0 PL=0
MOVL C01762 V=800.0 PL=0
MOVL C01763 V=800.0 PL=0
MOVL C01764 V=800.0 PL=0
MOVL C01765 V=800.0 PL=0
MOVL C01766 V=800.0 PL=0
MOVL C01767 V=800.0 PL=0
MOVL C01768 V=800.0 PL=0
MOVL C01769 V=800.0 PL=0
MOVL C01770 V=800.0 PL=0
MOVL C01771 V=800.0 PL=0
MOVL C01772 V=800.0 PL=0
MOVL C01773 V=800.0 PL=0
MOVL C01774 V=800.0 PL=0
MOVL C01775 V=800.0 PL=0
MOVL C01776 V=800.0 PL=0
MOVL C01777 V=800.0 PL=0
MOVL C01778 V=800.0 PL=0
MOVL C01779 V=800.0 PL=0
MOVL C01780 V=800.0 PL=0
MOVL C01781 V=800.0 PL=0
MOVL C01782 V=800.0 PL=0
MOVL C01783 V=800.0 PL=0
MOVL C01784 V=800.0 PL=0
MOVL C01785 V=800.0 PL=0
MOVL C01786 V=800.0 PL=0
MOVL C01787 V=800.0 PL=0
MOVL C01788 V=800.0 PL=0
MOVL C01789 V=800.0 PL=0
MOVL C01790 V=800.0 PL=0
MOVL C01791 V=800.0 PL=0
MOVL C01792 V=800.0 PL=0
MOVL C01793 V=800.0 PL=0
MOVL C01794 V=800.0 PL=0
MOVL C01795 V=800.0 PL=0
MOVL C01796 V=800.0 PL=0
MOVL C01797 V=800.0 PL=0
MOVL C01798 V=800.0 PL=0
MOVL C01799 V=800.0 PL=0
MOVL C01800 V=800.0 PL=0
MOVL C01801 V=800.0 PL=0
MOVL C01802 V=800.0 PL=0
MOVL C01803 V=800.0 PL=0
MOVL C01804 V=800.0 PL=0
MOVL C01805 V=800.0 PL=0
MOVL C01806 V=800.0 PL=0
MOVL C01807 V=800.0 PL=0
MOVL C01808 V=800.0 PL=0
MOVL C01809 V=800.0 PL=0
MOVL C01810 V=800.0 PL=0
MOVL C01811 V=800.0 PL=0
MOVL C01812 V=800.0 PL=0
MOVL C01813 V=800.0 PL=0
MOVL C01814 V=800.0 PL=0
MOVL C01815 V=800.0 PL=0
MOVL C01816 V=800.0 PL=0
MOVL C01817 V=800.0 PL=0
MOVL C01818 V=800.0 PL=0
MOVL C01819 V=800.0 PL=0
MOVL C01820 V=800.0 PL=0
MOVL C01821 V=800.0 PL=0
MOVL C01822 V=800.0 PL=0
MOVL C01823 V=800.0 PL=0
MOVL C01824 V=800.0 PL=0
MOVL C01825 V=800.0 PL=0
MOVL C01826 V=800.0 PL=0
MOVL C01827 V=800.0 PL=0
MOVL C01828 V=800.0 PL=0
MOVL C01829 V=800.0 PL=0
MOVL C01830 V=800.0 PL=0
MOVL C01831 V=800.0 PL=0
MOVL C01832 V=800.0 PL=0
MOVL C01833 V=800.0 PL=0
MOVL C01834 V=800.0 PL=0
MOVL C01835 V=800.0 PL=0
MOVL C01836 V=800.0 PL=0
MOVL C01837 V=800.0 PL=0
MOVL C01838 V=800.0 PL=0
MOVL C01839 V=800.0 PL=0
MOVL C01840 V=800.0 PL=0
MOVL C01841 V=800.0 PL=0
MOVL C01842 V=800.0 PL=0
MOVL C01843 V=800.0 PL=0
MOVL C01844 V=800.0 PL=0
MOVL C01845 V=800.0 PL=0
MOVL C01846 V=800.0 PL=0
MOVL C01847 V=800.0 PL=0
MOVL C01848 V=800.0 PL=0
MOVL C01849 V=800.0 PL=0
MOVL C01850 V=800.0 PL=0
MOVL C01851 V=800.0 PL=0
MOVL C01852 V=800.0 PL=0
MOVL C01853 V=800.0 PL=0
MOVL C01854 V=800.0 PL=0
MOVL C01855 V=800.0 PL=0
MOVL C01856 V=800.0 PL=0
MOVL C01857 V=800.0 PL=0
MOVL C01858 V=800.0 PL=0
MOVL C01859 V=800.0 PL=0
MOVL C01860 V=800.0 PL=0
MOVL C01861 V=800.0 PL=0
MOVL C01862 V=800.0 PL=0
MOVL C01863 V=800.0 PL=0
MOVL C01864 V=800.0 PL=0
MOVL C01865 V=800.0 PL=0
MOVL C01866 V=800.0 PL=0
MOVL C01867 V=800.0 PL=0
MOVL C01868 V=800.0 PL=0
MOVL C01869 V=800.0 PL=0
MOVL C01870 V=800.0 PL=0
MOVL C01871 V=800.0 PL=0
MOVL C01872 V=800.0 PL=0
MOVL C01873 V=800.0 PL=0
MOVL C01874 V=800.0 PL=0
MOVL C01875 V=800.0 PL=0
MOVL C01876 V=800.0 PL=0
MOVL C01877 V=800.0 PL=0
MOVL C01878 V=800.0 PL=0
MOVL C01879 V=800.0 PL=0
MOVL C01880 V=800.0 PL=0
MOVL C01881 V=800.0 PL=0
MOVL C01882 V=800.0 PL=0
MOVL C01883 V=800.0 PL=0
MOVL C01884 V=800.0 PL=0
MOVL C01885 V=800.0 PL=0
MOVL C01886 V=800.0 PL=0
MOVL C01887 V=800.0 PL=0
MOVL C01888 V=800.0 PL=0
MOVL C01889 V=800.0 PL=0
MOVL C01890 V=800.0 PL=0
MOVL C01891 V=800.0 PL=0
MOVL C01892 V=800.0 PL=0
MOVL C01893 V=800.0 PL=0
MOVL C01894 V=800.0 PL=0
MOVL C01895 V=800.0 PL=0
MOVL C01896 V=800.0 PL=0
MOVL C01897 V=800.0 PL=0
MOVL C01898 V=800.0 PL=0
MOVL C01899 V=800.0 PL=0
MOVL C01900 V=800.0 PL=0
MOVL C01901 V=800.0 PL=0
MOVL C01902 V=800.0 PL=0
MOVL C01903 V=800.0 PL=0
MOVL C01904 V=800.0 PL=0
MOVL C01905 V=800.0 PL=0
MOVL C01906 V=800.0 PL=0
MOVL C01907 V=800.0 PL=0
MOVL C01908 V=800.0 PL=0
MOVL C01909 V=800.0 PL=0
MOVL C01910 V=800.0 PL=0
MOVL C01911 V=800.0 PL=0
MOVL C01912 V=800.0 PL=0
MOVL C01913 V=800.0 PL=0
MOVL C01914 V=800.0 PL=0
MOVL C01915 V=800.0 PL=0
MOVL C01916 V=800.0 PL=0
MOVL C01917 V=800.0 PL=0
MOVL C01918 V=800.0 PL=0
MOVL C01919 V=800.0 PL=0
MOVL C01920 V=800.0 PL=0
MOVL C01921 V=800.0 PL=0
MOVL C01922 V=800.0 PL=0
MOVL C01923 V=800.0 PL=0
MOVL C01924 V=800.0 PL=0
MOVL C01925 V=800.0 PL=0
MOVL C01926 V=800.0 PL=0
MOVL C01927 V=800.0 PL=0
MOVL C01928 V=800.0 PL=0
MOVL C01929 V=800.0 PL=0
MOVL C01930 V=800.0 PL=0
MOVL C01931 V=800.0 PL=0
MOVL C01932 V=800.0 PL=0
MOVL C01933 V=800.0 PL=0
MOVL C01934 V=800.0 PL=0
MOVL C01935 V=800.0 PL=0
MOVL C01936 V=800.0 PL=0
MOVL C01937 V=800.0 PL=0
MOVL C01938 V=800.0 PL=0
MOVL C01939 V=800.0 PL=0
MOVL C01940 V=800.0 PL=0
MOVL C01941 V=800.0 PL=0
MOVL C01942 V=800.0 PL=0
MOVL C01943 V=800.0 PL=0
MOVL C01944 V=800.0 PL=0
MOVL C01945 V=800.0 PL=0
MOVL C01946 V=800.0 PL=0
MOVL C01947 V=800.0 PL=0
MOVL C01948 V=800.0 PL=0
MOVL C01949 V=800.0 PL=0
MOVL C01950 V=800.0 PL=0
MOVL C01951 V=800.0 PL=0
MOVL C01952 V=800.0 PL=0
MOVL C01953 V=800.0 PL=0
MOVL C01954 V=800.0 PL=0
MOVL C01955 V=800.0 PL=0
MOVL C01956 V=800.0 PL=0
MOVL C01957 V=800.0 PL=0
MOVL C01958 V=800.0 PL=0
MOVL C01959 V=800.0 PL=0
MOVL C01960 V=800.0 PL=0
MOVL C01961 V=800.0 PL=0
MOVL C01962 V=800.0 PL=0
MOVL C01963 V=800.0 PL=0
MOVL C01964 V=800.0 PL=0
MOVL C01965 V=800.0 PL=0
MOVL C01966 V=800.0 PL=0
MOVL C01967 V=800.0 PL=0
MOVL C01968 V=800.0 PL=0
MOVL C01969 V=800.0 PL=0
MOVL C01970 V=800.0 PL=0
MOVL C01971 V=800.0 PL=0
MOVL C01972 V=800.0 PL=0
MOVL C01973 V=800.0 PL=0
MOVL C01974 V=800.0 PL=0
MOVL C01975 V=800.0 PL=0
MOVL C01976 V=800.0 PL=0
MOVL C01977 V=800.0 PL=0
MOVL C01978 V=800.0 PL=0
MOVL C01979 V=800.0 PL=0
MOVL C01980 V=800.0 PL=0
MOVL C01981 V=800.0 PL=0
MOVL C01982 V=800.0 PL=0
MOVL C01983 V=800.0 PL=0
MOVL C01984 V=800.0 PL=0
MOVL C01985 V=800.0 PL=0
MOVL C01986 V=800.0 PL=0
MOVL C01987 V=800.0 PL=0
MOVL C01988 V=800.0 PL=0
MOVL C01989 V=800.0 PL=0
MOVL C01990 V=800.0 PL=0
MOVL C01991 V=800.0 PL=0
MOVL C01992 V=800.0 PL=0
MOVL C01993 V=800.0 PL=0
MOVL C01994 V=800.0 PL=0
MOVL C01995 V=800.0 PL=0
MOVL C01996 V=800.0 PL=0
MOVL C01997 V=800.0 PL=0
MOVL C01998 V=800.0 PL=0
MOVL C01999 V=800.0 PL=0
MOVL C02000 V=800.0 PL=0
MOVL C02001 V=800.0 PL=0
MOVL C02002 V=800.0 PL=0
MOVL C02003 V=800.0 PL=0
MOVL C02004 V=800.0 PL=0
MOVL C02005 V=800.0 PL=0
MOVL C02006 V=800.0 PL=0
MOVL C02007 V=800.0 PL=0
MOVL C02008 V=800.0 PL=0
MOVL C02009 V=800.0 PL=0
MOVL C02010 V=800.0 PL=0
MOVL C02011 V=800.0 PL=0
MOVL C02012 V=800.0 PL=0
MOVL C02013 V=800.0 PL=0
MOVL C02014 V=800.0 PL=0
MOVL C02015 V=800.0 PL=0
MOVL C02016 V=800.0 PL=0
MOVL C02017 V=800.0 PL=0
MOVL C02018 V=800.0 PL=0
MOVL C02019 V=800.0 PL=0
MOVL C02020 V=800.0 PL=0
MOVL C02021 V=800.0 PL=0
MOVL C02022 V=800.0 PL=0
MOVL C02023 V=800.0 PL=0
MOVL C02024 V=800.0 PL=0
MOVL C02025 V=800.0 PL=0
MOVL C02026 V=800.0 PL=0
MOVL C02027 V=800.0 PL=0
MOVL C02028 V=800.0 PL=0
MOVL C02029 V=800.0 PL=0
MOVL C02030 V=800.0 PL=0
MOVL C02031 V=800.0 PL=0
MOVL C02032 V=800.0 PL=0
MOVL C02033 V=800.0 PL=0
MOVL C02034 V=800.0 PL=0
MOVL C02035 V=800.0 PL=0
MOVL C02036 V=800.0 PL=0
MOVL C02037 V=800.0 PL=0
MOVL C02038 V=800.0 PL=0
MOVL C02039 V=800.0 PL=0
MOVL C02040 V=800.0 PL=0
MOVL C02041 V=800.0 PL=0
MOVL C02042 V=800.0 PL=0
MOVL C02043 V=800.0 PL=0
MOVL C02044 V=800.0 PL=0
MOVL C02045 V=800.0 PL=0
MOVL C02046 V=800.0 PL=0
MOVL C02047 V=800.0 PL=0
MOVL C02048 V=800.0 PL=0
MOVL C02049 V=800.0 PL=0
MOVL C02050 V=800.0 PL=0
MOVL C02051 V=800.0 PL=0
MOVL C02052 V=800.0 PL=0
MOVL C02053 V=800.0 PL=0
MOVL C02054 V=800.0 PL=0
MOVL C02055 V=800.0 PL=0
MOVL C02056 V=800.0 PL=0
MOVL C02057 V=800.0 PL=0
MOVL C02058 V=800.0 PL=0
